KUKA KRL program: EPS_2_25862_MH07_A_20251016035156.src

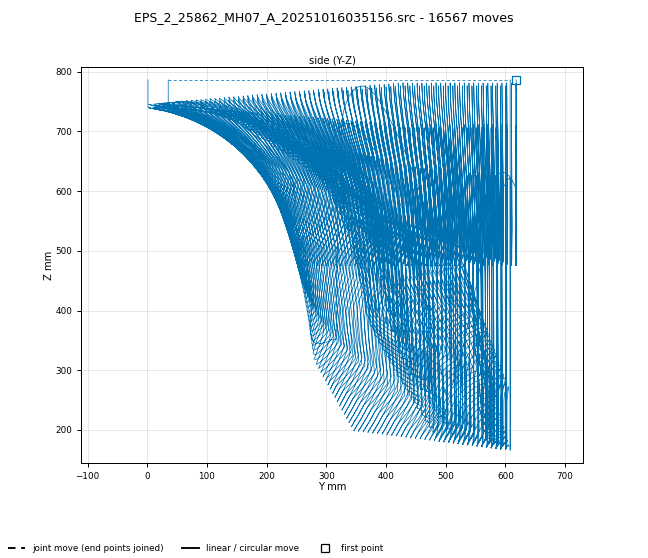
[picture p0: tool path of EPS_2_25862_MH07_A_20251016035156.src, 16567 of 16569 moves have a stored position in this frame; points joined in program order, loops and branches not executed]
&ACCESS RVP
&REL 4
&COMMENT QRS 19112012
&PARAM EDITMASK = *
DEF PART()
EXT BAS (BAS_COMMAND :IN,REAL :IN )
INT I
BAS (#INITMOV,0 )

;KUKA QRS Post kuka4.cps  Date:22-06-2017 !

File_ID=2887

QRS_PRE_INIT()

;Init var - Until changes are made in qrs_pre_init
Outlet_Square_prg=0
Inlet_1_Square_prg=0
Inlet_2_Square_prg=0
Inlet_3_Square_prg=0
Inlet_4_Square_prg=0
Inlet_5_Square_prg=0

Outlet_1={X 0.000, Y 425.000, Z 510.000, B 0.000, E1 0.000 }
Inlet_1={X 0.000, Y 529.170, Z 407.000, B 0.000, E1 90.000 }
Inlet_2={X 0.000, Y 425.000, Z 440.000, B 0.000, E1 163.000 }
Outlet_1_type=533
Inlet_1_type=299
Inlet_2_type=533
;QRS#1=Sidecore dimensions
;QRS#2=525-21" Concrete
;QRS#3=300-12" PVC SDR 35
;QRS#4=525-21" Concrete
;QRS#5=
;QRS#6=
;QRS#7=
;QRS#8=
;QRS#9=S306-32
;QRS#10=16M PSX
;QRS#11=S306-32
;QRS#12=
;QRS#13=
;QRS#14=
;QRS#15=
;QRS#16=1220x127x1143 3,75'
;QRS#17=EPS Height
;QRS#18=776,5
;QRS#19=*
;QRS#20= UPDATED VERSION 22-06-2017
;QRS#21=*
Outlet_Square=0250
Inlet_1_Square=0150
Inlet_2_Square=0250
Inlet_3_Square=0
Inlet_4_Square=0
Inlet_5_Square=0
Mill_Square=1
Outlet_Square_Prg=263
Inlet_1_Square_prg=206
Inlet_2_Square_prg=263

QRS_INIT()

$ADVANCE=5

; T1
PTP {E1 170.881,E2 170.881}
PTP {X 0,Y 617.976,A -85,B 0,C 180,E1 170.881,E2 170.881,E3 0,E4 0,E5 0,E6 0}
QRS_SPEED_INIT()
LIN {X 0,Y 617.976,Z 786.5,A -85,B 0,C 180,E1 170.881,E2 170.881,E3 0,E4 0,E5 0,E6 0} C_VEL
LIN {X 0,Y 617.976,Z 614.117,A -85,B 0,C 180,E1 170.881,E2 170.881} C_VEL
LIN {X 0,Y 617.976,Z 605.661,A -85,B 0,C 180,E1 170.881,E2 170.881} C_VEL
LIN {X 0,Y 617.953,Z 603.915,A -85,B 0,C 180,E1 171.157,E2 171.157} C_VEL
LIN {X 0,Y 617.982,Z 609.709,A -85,B 0,C 180,E1 172.119,E2 172.119} C_VEL
LIN {X 0,Y 617.938,Z 613.421,A -85,B 0,C 180,E1 172.818,E2 172.818} C_VEL
LIN {X 0,Y 617.912,Z 616.713,A -85,B 0,C 180,E1 173.515,E2 173.515} C_VEL
LIN {X 0,Y 617.958,Z 619.593,A -85,B 0,C 180,E1 174.213,E2 174.213} C_VEL
LIN {X 0,Y 617.989,Z 621.321,A -85,B 0,C 180,E1 174.678,E2 174.678} C_VEL
LIN {X 0,Y 617.915,Z 624.296,A -85,B 0,C 180,E1 175.605,E2 175.605} C_VEL
LIN {X 0,Y 617.888,Z 626.636,A -85,B 0,C 180,E1 176.531,E2 176.531} C_VEL
LIN {X 0,Y 617.975,Z 628.385,A -85,B 0,C 180,E1 177.457,E2 177.457} C_VEL
LIN {X 0,Y 617.924,Z 629.629,A -85,B 0,C 180,E1 178.382,E2 178.382} C_VEL
LIN {X 0,Y 617.892,Z 630.009,A -85,B 0,C 180,E1 178.844,E2 178.844} C_VEL
LIN {X 0,Y 617.918,Z 630.398,A -85,B 0,C 180,E1 179.769,E2 179.769} C_VEL
LIN {X 0,Y 617.987,Z 630.242,A -85,B 0,C 180,E1 180.693,E2 180.693} C_VEL
LIN {X 0,Y 617.941,Z 629.932,A -85,B 0,C 180,E1 181.156,E2 181.156} C_VEL
LIN {X 0,Y 617.883,Z 628.987,A -85,B 0,C 180,E1 182.08,E2 182.08} C_VEL
LIN {X 0,Y 617.888,Z 628.258,A -85,B 0,C 180,E1 182.543,E2 182.543} C_VEL
LIN {X 0,Y 617.984,Z 626.416,A -85,B 0,C 180,E1 183.468,E2 183.468} C_VEL
LIN {X 0,Y 617.908,Z 624.054,A -85,B 0,C 180,E1 184.395,E2 184.395} C_VEL
LIN {X 0,Y 617.895,Z 621.008,A -85,B 0,C 180,E1 185.323,E2 185.323} C_VEL
LIN {X 0,Y 617.935,Z 619.264,A -85,B 0,C 180,E1 185.787,E2 185.787} C_VEL
LIN {X 0,Y 617.983,Z 615.24,A -85,B 0,C 180,E1 186.716,E2 186.716} C_VEL
LIN {X 0,Y 617.925,Z 610.505,A -85,B 0,C 180,E1 187.649,E2 187.649} C_VEL
LIN {X 0,Y 617.962,Z 604.94,A -85,B 0,C 180,E1 188.595,E2 188.595} C_VEL
LIN {X 0,Y 618,Z 599.801,A -85,B 0,C 180,E1 189.355,E2 189.355} C_VEL
LIN {X 0,Y 617.956,Z 594.236,A -85,B 0,C 180,E1 190.089,E2 190.089} C_VEL
LIN {X 0,Y 617.957,Z 588.665,A -85,B 0,C 180,E1 190.75,E2 190.75} C_VEL
LIN {X 0,Y 617.996,Z 581.774,A -85,B 0,C 180,E1 191.486,E2 191.486} C_VEL
LIN {X 0,Y 617.98,Z 574.003,A -85,B 0,C 180,E1 192.224,E2 192.224} C_VEL
LIN {X 0,Y 617.981,Z 566.983,A -85,B 0,C 180,E1 192.815,E2 192.815} C_VEL
LIN {X 0,Y 618.01,Z 560.186,A -85,B 0,C 180,E1 193.334,E2 193.334} C_VEL
LIN {X 0,Y 618.026,Z 552.645,A -85,B 0,C 180,E1 193.853,E2 193.853} C_VEL
LIN {X 0,Y 618.025,Z 542.922,A -85,B 0,C 180,E1 194.449,E2 194.449} C_VEL
LIN {X 0,Y 617.99,Z 534.465,A -85,B 0,C 180,E1 194.898,E2 194.898} C_VEL
LIN {X 0,Y 618.023,Z 525.506,A -85,B 0,C 180,E1 195.313,E2 195.313} C_VEL
LIN {X 0,Y 618.026,Z 518.365,A -85,B 0,C 180,E1 195.605,E2 195.605} C_VEL
LIN {X 0,Y 617.977,Z 509.686,A -85,B 0,C 180,E1 195.915,E2 195.915} C_VEL
LIN {X 0,Y 617.998,Z 501.407,A -85,B 0,C 180,E1 196.165,E2 196.165} C_VEL
LIN {X 0,Y 618.025,Z 492.067,A -85,B 0,C 180,E1 196.398,E2 196.398} C_VEL
LIN {X 0,Y 617.952,Z 480.006,A -85,B 0,C 180,E1 196.626,E2 196.626} C_VEL
LIN {X 0,Y 617.88,Z 476.03,A -85,B 0,C 180,E1 196.691,E2 196.691} C_VEL
LIN {X 0,Y 618.007,Z 476.03,A -85,B 0,C 180,E1 196.801,E2 196.801} C_VEL
LIN {X 0,Y 617.96,Z 476.03,A -85,B 0,C 180,E1 200.048,E2 200.048} C_VEL
LIN {X 0,Y 617.455,Z 476.03,A -85,B 0,C 180,E1 202.548,E2 202.548} C_VEL
LIN {X 0,Y 617.918,Z 476.03,A -85,B 0,C 180,E1 205.056,E2 205.056} C_VEL
LIN {X 0,Y 617.406,Z 476.03,A -85,B 0,C 180,E1 207.66,E2 207.66} C_VEL
LIN {X 0,Y 617.848,Z 476.03,A -85,B 0,C 180,E1 210.28,E2 210.28} C_VEL
LIN {X 0,Y 617.31,Z 476.03,A -85,B 0,C 180,E1 213.027,E2 213.027} C_VEL
LIN {X 0,Y 617.797,Z 476.03,A -85,B 0,C 180,E1 215.799,E2 215.799} C_VEL
LIN {X 0,Y 617.573,Z 476.03,A -85,B 0,C 180,E1 218.099,E2 218.099} C_VEL
LIN {X 0,Y 617.553,Z 476.03,A -85,B 0,C 180,E1 218.722,E2 218.722} C_VEL
LIN {X 0,Y 617.792,Z 476.03,A -85,B 0,C 180,E1 221.731,E2 221.731} C_VEL
LIN {X 0,Y 617.879,Z 476.03,A -85,B 0,C 180,E1 225.099,E2 225.099} C_VEL
LIN {X 0,Y 617.456,Z 476.03,A -85,B 0,C 180,E1 228.308,E2 228.308} C_VEL
LIN {X 0,Y 617.797,Z 476.03,A -85,B 0,C 180,E1 231.296,E2 231.296} C_VEL
LIN {X 0,Y 617.723,Z 476.03,A -85,B 0,C 180,E1 235.802,E2 235.802} C_VEL
LIN {X 0,Y 617.906,Z 476.03,A -85,B 0,C 180,E1 237.009,E2 237.009} C_VEL
LIN {X 0,Y 617.905,Z 476.03,A -85,B 0,C 180,E1 240.133,E2 240.133} C_VEL
LIN {X 0,Y 617.607,Z 476.03,A -85,B 0,C 180,E1 240.837,E2 240.837} C_VEL
LIN {X 0,Y 617.093,Z 483.978,A -85,B 0,C 180,E1 241.034,E2 241.034} C_VEL
LIN {X 0,Y 617.595,Z 516.166,A -85,B 0,C 180,E1 241.478,E2 241.478} C_VEL
LIN {X 0,Y 617.687,Z 536.067,A -85,B 0,C 180,E1 241.783,E2 241.783} C_VEL
LIN {X 0,Y 617.745,Z 546.864,A -85,B 0,C 180,E1 242.005,E2 242.005} C_VEL
LIN {X 0,Y 617.719,Z 563.319,A -85,B 0,C 180,E1 242.427,E2 242.427} C_VEL
LIN {X 0,Y 617.856,Z 576.645,A -85,B 0,C 180,E1 242.85,E2 242.85} C_VEL
LIN {X 0,Y 617.886,Z 587.938,A -85,B 0,C 180,E1 243.257,E2 243.257} C_VEL
LIN {X 0,Y 617.754,Z 601.563,A -85,B 0,C 180,E1 243.815,E2 243.815} C_VEL
LIN {X 0,Y 617.879,Z 613.583,A -85,B 0,C 180,E1 244.383,E2 244.383} C_VEL
LIN {X 0,Y 617.884,Z 625.767,A -85,B 0,C 180,E1 245.021,E2 245.021} C_VEL
LIN {X 0,Y 617.847,Z 637.421,A -85,B 0,C 180,E1 245.696,E2 245.696} C_VEL
LIN {X 0,Y 617.908,Z 648.138,A -85,B 0,C 180,E1 246.38,E2 246.38} C_VEL
LIN {X 0,Y 617.924,Z 659.39,A -85,B 0,C 180,E1 247.168,E2 247.168} C_VEL
LIN {X 0,Y 617.915,Z 669.503,A -85,B 0,C 180,E1 247.938,E2 247.938} C_VEL
LIN {X 0,Y 617.885,Z 680.645,A -85,B 0,C 180,E1 248.869,E2 248.869} C_VEL
LIN {X 0,Y 617.922,Z 690.764,A -85,B 0,C 180,E1 249.797,E2 249.797} C_VEL
LIN {X 0,Y 617.932,Z 699.516,A -85,B 0,C 180,E1 250.667,E2 250.667} C_VEL
LIN {X 0,Y 617.881,Z 706.64,A -85,B 0,C 180,E1 251.422,E2 251.422} C_VEL
LIN {X 0,Y 617.901,Z 715.015,A -85,B 0,C 180,E1 252.391,E2 252.391} C_VEL
LIN {X 0,Y 617.982,Z 723.19,A -85,B 0,C 180,E1 253.428,E2 253.428} C_VEL
LIN {X 0,Y 617.837,Z 731.707,A -85,B 0,C 180,E1 254.61,E2 254.61} C_VEL
LIN {X 0,Y 617.891,Z 738.767,A -85,B 0,C 180,E1 255.697,E2 255.697} C_VEL
LIN {X 0,Y 617.963,Z 744.12,A -85,B 0,C 180,E1 256.591,E2 256.591} C_VEL
LIN {X 0,Y 617.785,Z 750.562,A -85,B 0,C 180,E1 257.772,E2 257.772} C_VEL
LIN {X 0,Y 617.806,Z 756.245,A -85,B 0,C 180,E1 258.953,E2 258.953} C_VEL
LIN {X 0,Y 617.974,Z 760.457,A -85,B 0,C 180,E1 259.949,E2 259.949} C_VEL
LIN {X 0,Y 617.8,Z 765.453,A -85,B 0,C 180,E1 261.249,E2 261.249} C_VEL
LIN {X 0,Y 617.8,Z 769.018,A -85,B 0,C 180,E1 262.35,E2 262.35} C_VEL
LIN {X 0,Y 617.952,Z 772.841,A -85,B 0,C 180,E1 263.748,E2 263.748} C_VEL
LIN {X 0,Y 617.735,Z 775.904,A -85,B 0,C 180,E1 265.14,E2 265.14} C_VEL
LIN {X 0,Y 617.832,Z 778.096,A -85,B 0,C 180,E1 266.531,E2 266.531} C_VEL
LIN {X 0,Y 617.874,Z 779.552,A -85,B 0,C 180,E1 267.919,E2 267.919} C_VEL
LIN {X 0,Y 617.748,Z 780.216,A -85,B 0,C 180,E1 268.844,E2 268.844} C_VEL
LIN {X 0,Y 617.993,Z 780.149,A -85,B 0,C 180,E1 271.155,E2 271.155} C_VEL
LIN {X 0,Y 617.921,Z 779.182,A -85,B 0,C 180,E1 272.543,E2 272.543} C_VEL
LIN {X 0,Y 617.992,Z 778.053,A -85,B 0,C 180,E1 273.468,E2 273.468} C_VEL
LIN {X 0,Y 617.764,Z 775.897,A -85,B 0,C 180,E1 274.86,E2 274.86} C_VEL
LIN {X 0,Y 617.792,Z 772.883,A -85,B 0,C 180,E1 276.253,E2 276.253} C_VEL
LIN {X 0,Y 617.96,Z 770.333,A -85,B 0,C 180,E1 277.182,E2 277.182} C_VEL
LIN {X 0,Y 617.863,Z 767.502,A -85,B 0,C 180,E1 278.116,E2 278.116} C_VEL
LIN {X 0,Y 617.789,Z 765.164,A -85,B 0,C 180,E1 278.829,E2 278.829} C_VEL
LIN {X 0,Y 617.862,Z 760.497,A -85,B 0,C 180,E1 280.05,E2 280.05} C_VEL
LIN {X 0,Y 617.967,Z 756.211,A -85,B 0,C 180,E1 281.044,E2 281.044} C_VEL
LIN {X 0,Y 617.792,Z 750.562,A -85,B 0,C 180,E1 282.227,E2 282.227} C_VEL
LIN {X 0,Y 617.814,Z 744.15,A -85,B 0,C 180,E1 283.412,E2 283.412} C_VEL
LIN {X 0,Y 617.958,Z 736.918,A -85,B 0,C 180,E1 284.6,E2 284.6} C_VEL
LIN {X 0,Y 617.812,Z 729.351,A -85,B 0,C 180,E1 285.734,E2 285.734} C_VEL
LIN {X 0,Y 617.84,Z 722.479,A -85,B 0,C 180,E1 286.674,E2 286.674} C_VEL
LIN {X 0,Y 617.977,Z 713.931,A -85,B 0,C 180,E1 287.734,E2 287.734} C_VEL
LIN {X 0,Y 617.889,Z 704.471,A -85,B 0,C 180,E1 288.81,E2 288.81} C_VEL
LIN {X 0,Y 617.892,Z 695.989,A -85,B 0,C 180,E1 289.695,E2 289.695} C_VEL
LIN {X 0,Y 617.937,Z 687.527,A -85,B 0,C 180,E1 290.511,E2 290.511} C_VEL
LIN {X 0,Y 617.894,Z 677.03,A -85,B 0,C 180,E1 291.44,E2 291.44} C_VEL
LIN {X 0,Y 617.882,Z 667.492,A -85,B 0,C 180,E1 292.219,E2 292.219} C_VEL
LIN {X 0,Y 617.9,Z 657.417,A -85,B 0,C 180,E1 292.976,E2 292.976} C_VEL
LIN {X 0,Y 617.911,Z 645.135,A -85,B 0,C 180,E1 293.813,E2 293.813} C_VEL
LIN {X 0,Y 617.904,Z 633.893,A -85,B 0,C 180,E1 294.512,E2 294.512} C_VEL
LIN {X 0,Y 617.836,Z 622.881,A -85,B 0,C 180,E1 295.139,E2 295.139} C_VEL
LIN {X 0,Y 617.892,Z 610.287,A -85,B 0,C 180,E1 295.776,E2 295.776} C_VEL
LIN {X 0,Y 617.876,Z 597.865,A -85,B 0,C 180,E1 296.34,E2 296.34} C_VEL
LIN {X 0,Y 617.703,Z 584.662,A -85,B 0,C 180,E1 296.873,E2 296.873} C_VEL
LIN {X 0,Y 617.832,Z 571.391,A -85,B 0,C 180,E1 297.323,E2 297.323} C_VEL
LIN {X 0,Y 617.741,Z 558.539,A -85,B 0,C 180,E1 297.705,E2 297.705} C_VEL
LIN {X 0,Y 617.713,Z 550.591,A -85,B 0,C 180,E1 297.907,E2 297.907} C_VEL
LIN {X 0,Y 617.901,Z 535.737,A -85,B 0,C 180,E1 298.213,E2 298.213} C_VEL
LIN {X 0,Y 617.756,Z 515.651,A -85,B 0,C 180,E1 298.521,E2 298.521} C_VEL
LIN {X 0,Y 617.026,Z 476.03,A -85,B 0,C 180,E1 299.084,E2 299.084} C_VEL
LIN {X 0,Y 618.06,Z 476.03,A -85,B 0,C 180,E1 299.464,E2 299.464} C_VEL
LIN {X 0,Y 618.044,Z 476.03,A -85,B 0,C 180,E1 300.269,E2 300.269} C_VEL
LIN {X 0,Y 617.372,Z 476.03,A -85,B 0,C 180,E1 304.15,E2 304.15} C_VEL
LIN {X 0,Y 617.829,Z 476.03,A -85,B 0,C 180,E1 305.797,E2 305.797} C_VEL
LIN {X 0,Y 617.555,Z 476.03,A -85,B 0,C 180,E1 308.721,E2 308.721} C_VEL
LIN {X 0,Y 617.763,Z 476.03,A -85,B 0,C 180,E1 311.733,E2 311.733} C_VEL
LIN {X 0,Y 617.85,Z 476.03,A -85,B 0,C 180,E1 315.097,E2 315.097} C_VEL
LIN {X 0,Y 617.449,Z 476.03,A -85,B 0,C 180,E1 318.308,E2 318.308} C_VEL
LIN {X 0,Y 617.792,Z 476.03,A -85,B 0,C 180,E1 321.296,E2 321.296} C_VEL
LIN {X 0,Y 617.737,Z 476.03,A -85,B 0,C 180,E1 325.799,E2 325.799} C_VEL
LIN {X 0,Y 617.89,Z 476.03,A -85,B 0,C 180,E1 327.008,E2 327.008} C_VEL
LIN {X 0,Y 617.613,Z 476.03,A -85,B 0,C 180,E1 330.18,E2 330.18} C_VEL
LIN {X 0,Y 617.623,Z 476.03,A -85,B 0,C 180,E1 332.351,E2 332.351} C_VEL
LIN {X 0,Y 617.512,Z 476.03,A -85,B 0,C 180,E1 335.243,E2 335.243} C_VEL
LIN {X 0,Y 617.738,Z 476.03,A -85,B 0,C 180,E1 337.463,E2 337.463} C_VEL
LIN {X 0,Y 617.768,Z 476.03,A -85,B 0,C 180,E1 341.452,E2 341.452} C_VEL
LIN {X 0,Y 617.981,Z 476.03,A -85,B 0,C 180,E1 342.394,E2 342.394} C_VEL
LIN {X 0,Y 618.01,Z 476.03,A -85,B 0,C 180,E1 347.185,E2 347.185} C_VEL
LIN {X 0,Y 617.973,Z 476.03,A -85,B 0,C 180,E1 351.885,E2 351.885} C_VEL
LIN {X 0,Y 618.058,Z 476.03,A -85,B 0,C 180,E1 356.532,E2 356.532} C_VEL
LIN {X 0,Y 618.062,Z 476.03,A -85,B 0,C 180,E1 361.155,E2 361.155} C_VEL
LIN {X 0,Y 618.025,Z 476.03,A -85,B 0,C 180,E1 365.786,E2 365.786} C_VEL
LIN {X 0,Y 618.005,Z 476.03,A -85,B 0,C 180,E1 370.456,E2 370.456} C_VEL
LIN {X 0,Y 617.94,Z 476.03,A -85,B 0,C 180,E1 375.198,E2 375.198} C_VEL
LIN {X 0,Y 617.959,Z 476.03,A -85,B 0,C 180,E1 380.048,E2 380.048} C_VEL
LIN {X 0,Y 617.477,Z 476.03,A -85,B 0,C 180,E1 382.547,E2 382.547} C_VEL
LIN {X 0,Y 617.928,Z 476.03,A -85,B 0,C 180,E1 385.055,E2 385.055} C_VEL
LIN {X 0,Y 617.434,Z 476.03,A -85,B 0,C 180,E1 387.658,E2 387.658} C_VEL
LIN {X 0,Y 617.899,Z 476.03,A -85,B 0,C 180,E1 390.277,E2 390.277} C_VEL
LIN {X 0,Y 617.363,Z 476.03,A -85,B 0,C 180,E1 393.024,E2 393.024} C_VEL
LIN {X 0,Y 617.83,Z 476.03,A -85,B 0,C 180,E1 395.797,E2 395.797} C_VEL
LIN {X 0,Y 617.922,Z 476.03,A -85,B 0,C 180,E1 398.694,E2 398.694} C_VEL
LIN {X 0,Y 617.441,Z 476.03,A -85,B 0,C 180,E1 401.76,E2 401.76} C_VEL
LIN {X 0,Y 617.884,Z 476.03,A -85,B 0,C 180,E1 404.9,E2 404.9} C_VEL
LIN {X 0,Y 617.788,Z 476.03,A -85,B 0,C 180,E1 408.273,E2 408.273} C_VEL
LIN {X 0,Y 617.543,Z 476.03,A -85,B 0,C 180,E1 411.278,E2 411.278} C_VEL
LIN {X 0,Y 617.56,Z 476.03,A -85,B 0,C 180,E1 411.902,E2 411.902} C_VEL
LIN {X 0,Y 617.774,Z 476.03,A -85,B 0,C 180,E1 414.199,E2 414.199} C_VEL
LIN {X 0,Y 617.311,Z 476.03,A -85,B 0,C 180,E1 416.973,E2 416.973} C_VEL
LIN {X 0,Y 617.85,Z 476.03,A -85,B 0,C 180,E1 419.72,E2 419.72} C_VEL
LIN {X 0,Y 617.406,Z 476.03,A -85,B 0,C 180,E1 422.341,E2 422.341} C_VEL
LIN {X 0,Y 617.916,Z 476.03,A -85,B 0,C 180,E1 424.944,E2 424.944} C_VEL
LIN {X 0,Y 617.454,Z 476.03,A -85,B 0,C 180,E1 427.452,E2 427.452} C_VEL
LIN {X 0,Y 617.947,Z 476.03,A -85,B 0,C 180,E1 429.952,E2 429.952} C_VEL
LIN {X 0,Y 617.716,Z 476.03,A -85,B 0,C 180,E1 432.386,E2 432.386} C_VEL
LIN {X 0,Y 617.639,Z 476.03,A -85,B 0,C 180,E1 434.795,E2 434.795} C_VEL
LIN {X 0,Y 617.816,Z 476.03,A -85,B 0,C 180,E1 437.834,E2 437.834} C_VEL
LIN {X 0,Y 617.958,Z 476.03,A -85,B 0,C 180,E1 438.667,E2 438.667} C_VEL
LIN {X 0,Y 617.118,Z 476.03,A -85,B 0,C 180,E1 438.912,E2 438.912} C_VEL
LIN {X 0,Y 617.601,Z 477.618,A -85,B 0,C 180,E1 438.969,E2 438.969} C_VEL
LIN {X 0,Y 617.721,Z 492.547,A -85,B 0,C 180,E1 439.358,E2 439.358} C_VEL
LIN {X 0,Y 617.858,Z 505.819,A -85,B 0,C 180,E1 439.776,E2 439.776} C_VEL
LIN {X 0,Y 617.814,Z 518.782,A -85,B 0,C 180,E1 440.243,E2 440.243} C_VEL
LIN {X 0,Y 617.844,Z 529.089,A -85,B 0,C 180,E1 440.664,E2 440.664} C_VEL
LIN {X 0,Y 617.915,Z 543.28,A -85,B 0,C 180,E1 441.324,E2 441.324} C_VEL
LIN {X 0,Y 617.87,Z 556.214,A -85,B 0,C 180,E1 442.001,E2 442.001} C_VEL
LIN {X 0,Y 617.891,Z 568.182,A -85,B 0,C 180,E1 442.701,E2 442.701} C_VEL
LIN {X 0,Y 617.899,Z 579.063,A -85,B 0,C 180,E1 443.399,E2 443.399} C_VEL
LIN {X 0,Y 617.912,Z 590.579,A -85,B 0,C 180,E1 444.213,E2 444.213} C_VEL
LIN {X 0,Y 617.9,Z 601.106,A -85,B 0,C 180,E1 445.025,E2 445.025} C_VEL
LIN {X 0,Y 617.886,Z 610.785,A -85,B 0,C 180,E1 445.837,E2 445.837} C_VEL
LIN {X 0,Y 617.945,Z 619.692,A -85,B 0,C 180,E1 446.648,E2 446.648} C_VEL
LIN {X 0,Y 617.931,Z 629.056,A -85,B 0,C 180,E1 447.573,E2 447.573} C_VEL
LIN {X 0,Y 617.868,Z 637.688,A -85,B 0,C 180,E1 448.498,E2 448.498} C_VEL
LIN {X 0,Y 617.917,Z 644.688,A -85,B 0,C 180,E1 449.307,E2 449.307} C_VEL
LIN {X 0,Y 617.934,Z 653.784,A -85,B 0,C 180,E1 450.462,E2 450.462} C_VEL
LIN {X 0,Y 617.824,Z 660.536,A -85,B 0,C 180,E1 451.387,E2 451.387} C_VEL
LIN {X 0,Y 617.897,Z 668.115,A -85,B 0,C 180,E1 452.543,E2 452.543} C_VEL
LIN {X 0,Y 617.949,Z 673.665,A -85,B 0,C 180,E1 453.469,E2 453.469} C_VEL
LIN {X 0,Y 617.77,Z 681.208,A -85,B 0,C 180,E1 454.86,E2 454.86} C_VEL
LIN {X 0,Y 617.862,Z 686.708,A -85,B 0,C 180,E1 456.02,E2 456.02} C_VEL
LIN {X 0,Y 617.963,Z 689.656,A -85,B 0,C 180,E1 456.717,E2 456.717} C_VEL
LIN {X 0,Y 617.838,Z 693.365,A -85,B 0,C 180,E1 457.65,E2 457.65} C_VEL
LIN {X 0,Y 617.773,Z 696.469,A -85,B 0,C 180,E1 458.508,E2 458.508} C_VEL
LIN {X 0,Y 617.884,Z 700.002,A -85,B 0,C 180,E1 459.641,E2 459.641} C_VEL
LIN {X 0,Y 617.973,Z 702.167,A -85,B 0,C 180,E1 460.456,E2 460.456} C_VEL
LIN {X 0,Y 617.795,Z 704.937,A -85,B 0,C 180,E1 461.637,E2 461.637} C_VEL
LIN {X 0,Y 617.827,Z 707.092,A -85,B 0,C 180,E1 462.819,E2 462.819} C_VEL
LIN {X 0,Y 617.971,Z 708.672,A -85,B 0,C 180,E1 464.004,E2 464.004} C_VEL
LIN {X 0,Y 617.751,Z 709.818,A -85,B 0,C 180,E1 465.203,E2 465.203} C_VEL
LIN {X 0,Y 617.724,Z 710.336,A -85,B 0,C 180,E1 466.313,E2 466.313} C_VEL
LIN {X 0,Y 617.943,Z 710.275,A -85,B 0,C 180,E1 467.607,E2 467.607} C_VEL
LIN {X 0,Y 617.891,Z 709.834,A -85,B 0,C 180,E1 468.632,E2 468.632} C_VEL
LIN {X 0,Y 617.915,Z 708.516,A -85,B 0,C 180,E1 470.05,E2 470.05} C_VEL
LIN {X 0,Y 617.852,Z 706.755,A -85,B 0,C 180,E1 471.287,E2 471.287} C_VEL
LIN {X 0,Y 617.777,Z 705.727,A -85,B 0,C 180,E1 471.911,E2 471.911} C_VEL
LIN {X 0,Y 617.771,Z 703.259,A -85,B 0,C 180,E1 473.047,E2 473.047} C_VEL
LIN {X 0,Y 617.987,Z 699.619,A -85,B 0,C 180,E1 474.399,E2 474.399} C_VEL
LIN {X 0,Y 617.775,Z 695.478,A -85,B 0,C 180,E1 475.702,E2 475.702} C_VEL
LIN {X 0,Y 617.81,Z 690.576,A -85,B 0,C 180,E1 476.99,E2 476.99} C_VEL
LIN {X 0,Y 617.965,Z 685.729,A -85,B 0,C 180,E1 478.104,E2 478.104} C_VEL
LIN {X 0,Y 617.824,Z 680.253,A -85,B 0,C 180,E1 479.241,E2 479.241} C_VEL
LIN {X 0,Y 617.876,Z 673.662,A -85,B 0,C 180,E1 480.446,E2 480.446} C_VEL
LIN {X 0,Y 617.958,Z 666.474,A -85,B 0,C 180,E1 481.621,E2 481.621} C_VEL
LIN {X 0,Y 617.833,Z 658.598,A -85,B 0,C 180,E1 482.791,E2 482.791} C_VEL
LIN {X 0,Y 617.908,Z 651.168,A -85,B 0,C 180,E1 483.79,E2 483.79} C_VEL
LIN {X 0,Y 617.983,Z 644.312,A -85,B 0,C 180,E1 484.645,E2 484.645} C_VEL
LIN {X 0,Y 617.871,Z 634.198,A -85,B 0,C 180,E1 485.795,E2 485.795} C_VEL
LIN {X 0,Y 617.907,Z 625.412,A -85,B 0,C 180,E1 486.706,E2 486.706} C_VEL
LIN {X 0,Y 617.936,Z 616.132,A -85,B 0,C 180,E1 487.591,E2 487.591} C_VEL
LIN {X 0,Y 617.914,Z 608.131,A -85,B 0,C 180,E1 488.304,E2 488.304} C_VEL
LIN {X 0,Y 617.888,Z 597.463,A -85,B 0,C 180,E1 489.176,E2 489.176} C_VEL
LIN {X 0,Y 617.868,Z 587.152,A -85,B 0,C 180,E1 489.95,E2 489.95} C_VEL
LIN {X 0,Y 617.904,Z 576.246,A -85,B 0,C 180,E1 490.699,E2 490.699} C_VEL
LIN {X 0,Y 617.902,Z 564.345,A -85,B 0,C 180,E1 491.441,E2 491.441} C_VEL
LIN {X 0,Y 617.813,Z 551.969,A -85,B 0,C 180,E1 492.142,E2 492.142} C_VEL
LIN {X 0,Y 617.871,Z 540.321,A -85,B 0,C 180,E1 492.731,E2 492.731} C_VEL
LIN {X 0,Y 617.851,Z 528.459,A -85,B 0,C 180,E1 493.271,E2 493.271} C_VEL
LIN {X 0,Y 617.723,Z 515.883,A -85,B 0,C 180,E1 493.784,E2 493.784} C_VEL
LIN {X 0,Y 617.856,Z 501.446,A -85,B 0,C 180,E1 494.275,E2 494.275} C_VEL
LIN {X 0,Y 617.787,Z 488.688,A -85,B 0,C 180,E1 494.654,E2 494.654} C_VEL
LIN {X 0,Y 617.518,Z 476.03,A -85,B 0,C 180,E1 494.988,E2 494.988} C_VEL
LIN {X 0,Y 618.002,Z 476.03,A -85,B 0,C 180,E1 495.111,E2 495.111} C_VEL
LIN {X 0,Y 617.354,Z 476.03,A -85,B 0,C 180,E1 498.318,E2 498.318} C_VEL
LIN {X 0,Y 617.788,Z 476.03,A -85,B 0,C 180,E1 501.296,E2 501.296} C_VEL
LIN {X 0,Y 617.711,Z 476.03,A -85,B 0,C 180,E1 505.803,E2 505.803} C_VEL
LIN {X 0,Y 617.878,Z 476.03,A -85,B 0,C 180,E1 507.007,E2 507.007} C_VEL
LIN {X 0,Y 618.031,Z 476.03,A -85,B 0,C 180,E1 511.492,E2 511.492} C_VEL
LIN {X 0,Y 617.378,Z 476.03,A -85,B 0,C 180,E1 515.271,E2 515.271} C_VEL
LIN {X 0,Y 617.928,Z 476.03,A -85,B 0,C 180,E1 517.47,E2 517.47} C_VEL
LIN {X 0,Y 618.059,Z 476.03,A -85,B 0,C 180,E1 522.8,E2 522.8} C_VEL
LIN {X 0,Y 616.384,Z 476.03,A -85,B 0,C 180,E1 523.155,E2 523.155} C_VEL
LIN {X 0,Y 616.161,Z 476.1,A -85,B 0,C 180,E1 523.179,E2 523.179} C_VEL
LIN {X 0,Y 617.345,Z 479.078,A -85,B 0,C 180,E1 523.254,E2 523.254} C_VEL
LIN {X 0,Y 617.909,Z 482.221,A -85,B 0,C 180,E1 523.316,E2 523.316} C_VEL
LIN {X 0,Y 617.987,Z 492.727,A -85,B 0,C 180,E1 523.526,E2 523.526} C_VEL
LIN {X 0,Y 617.947,Z 501.655,A -85,B 0,C 180,E1 523.751,E2 523.751} C_VEL
LIN {X 0,Y 617.991,Z 509.87,A -85,B 0,C 180,E1 524.001,E2 524.001} C_VEL
LIN {X 0,Y 617.968,Z 518.24,A -85,B 0,C 180,E1 524.299,E2 524.299} C_VEL
LIN {X 0,Y 617.97,Z 524.958,A -85,B 0,C 180,E1 524.572,E2 524.572} C_VEL
LIN {X 0,Y 618.003,Z 533.233,A -85,B 0,C 180,E1 524.953,E2 524.953} C_VEL
LIN {X 0,Y 618.025,Z 541.829,A -85,B 0,C 180,E1 525.402,E2 525.402} C_VEL
LIN {X 0,Y 617.985,Z 551.76,A -85,B 0,C 180,E1 525.997,E2 525.997} C_VEL
LIN {X 0,Y 618,Z 559.381,A -85,B 0,C 180,E1 526.518,E2 526.518} C_VEL
LIN {X 0,Y 618.006,Z 566.245,A -85,B 0,C 180,E1 527.037,E2 527.037} C_VEL
LIN {X 0,Y 618.001,Z 573.331,A -85,B 0,C 180,E1 527.629,E2 527.629} C_VEL
LIN {X 0,Y 617.98,Z 581.22,A -85,B 0,C 180,E1 528.367,E2 528.367} C_VEL
LIN {X 0,Y 617.981,Z 586.842,A -85,B 0,C 180,E1 528.956,E2 528.956} C_VEL
LIN {X 0,Y 618.011,Z 591.964,A -85,B 0,C 180,E1 529.544,E2 529.544} C_VEL
LIN {X 0,Y 617.972,Z 597.992,A -85,B 0,C 180,E1 530.31,E2 530.31} C_VEL
LIN {X 0,Y 617.938,Z 603.365,A -85,B 0,C 180,E1 531.075,E2 531.075} C_VEL
LIN {X 0,Y 617.953,Z 603.915,A -85,B 0,C 180,E1 531.157,E2 531.157} C_VEL
LIN {X 0,Y 614.025,Z 612.896,A -85,B 0,C 180,E1 532.531,E2 532.531} C_VEL
LIN {X 0,Y 610.136,Z 619.876,A -85,B 0,C 180,E1 533.98,E2 533.98} C_VEL
LIN {X 0,Y 610.076,Z 627.528,A -85,B 0,C 180,E1 536.441,E2 536.441} C_VEL
LIN {X 0,Y 610.102,Z 630.881,A -85,B 0,C 180,E1 538.576,E2 538.576} C_VEL
LIN {X 0,Y 610.104,Z 630.818,A -85,B 0,C 180,E1 541.42,E2 541.42} C_VEL
LIN {X 0,Y 610.115,Z 625.509,A -85,B 0,C 180,E1 544.267,E2 544.267} C_VEL
LIN {X 0,Y 610.138,Z 614.506,A -85,B 0,C 180,E1 547.125,E2 547.125} C_VEL
LIN {X 0,Y 610.2,Z 597.879,A -85,B 0,C 180,E1 549.819,E2 549.819} C_VEL
LIN {X 0,Y 610.219,Z 576.647,A -85,B 0,C 180,E1 552.172,E2 552.172} C_VEL
LIN {X 0,Y 610.331,Z 550.663,A -85,B 0,C 180,E1 554.177,E2 554.177} C_VEL
LIN {X 0,Y 610.405,Z 521.112,A -85,B 0,C 180,E1 555.702,E2 555.702} C_VEL
LIN {X 0,Y 610.453,Z 489.709,A -85,B 0,C 180,E1 556.662,E2 556.662} C_VEL
LIN {X 0,Y 610.085,Z 476.03,A -85,B 0,C 180,E1 556.951,E2 556.951} C_VEL
LIN {X 0,Y 609.583,Z 476.03,A -85,B 0,C 180,E1 561.871,E2 561.871} C_VEL
LIN {X 0,Y 610.001,Z 476.03,A -85,B 0,C 180,E1 564.954,E2 564.954} C_VEL
LIN {X 0,Y 609.766,Z 476.03,A -85,B 0,C 180,E1 569.772,E2 569.772} C_VEL
LIN {X 0,Y 609.713,Z 476.03,A -85,B 0,C 180,E1 576.578,E2 576.578} C_VEL
LIN {X 0,Y 609.798,Z 476.03,A -85,B 0,C 180,E1 582.091,E2 582.091} C_VEL
LIN {X 0,Y 609.521,Z 476.03,A -85,B 0,C 180,E1 587.878,E2 587.878} C_VEL
LIN {X 0,Y 609.49,Z 476.03,A -85,B 0,C 180,E1 592.642,E2 592.642} C_VEL
LIN {X 0,Y 609.897,Z 476.03,A -85,B 0,C 180,E1 597.562,E2 597.562} C_VEL
LIN {X 0,Y 609.828,Z 476.03,A -85,B 0,C 180,E1 600.533,E2 600.533} C_VEL
LIN {X 0,Y 610.755,Z 548.666,A -85,B 0,C 180,E1 601.697,E2 601.697} C_VEL
LIN {X 0,Y 610.747,Z 588.608,A -85,B 0,C 180,E1 602.946,E2 602.946} C_VEL
LIN {X 0,Y 610.579,Z 625.307,A -85,B 0,C 180,E1 604.674,E2 604.674} C_VEL
LIN {X 0,Y 610.427,Z 661.111,A -85,B 0,C 180,E1 607.004,E2 607.004} C_VEL
LIN {X 0,Y 610.29,Z 692.229,A -85,B 0,C 180,E1 609.675,E2 609.675} C_VEL
LIN {X 0,Y 610.174,Z 719.223,A -85,B 0,C 180,E1 612.676,E2 612.676} C_VEL
LIN {X 0,Y 610.128,Z 742.058,A -85,B 0,C 180,E1 615.997,E2 615.997} C_VEL
LIN {X 0,Y 610.103,Z 760.364,A -85,B 0,C 180,E1 619.634,E2 619.634} C_VEL
LIN {X 0,Y 610.018,Z 772.184,A -85,B 0,C 180,E1 623.084,E2 623.084} C_VEL
LIN {X 0,Y 609.94,Z 777.931,A -85,B 0,C 180,E1 625.729,E2 625.729} C_VEL
LIN {X 0,Y 609.966,Z 781.082,A -85,B 0,C 180,E1 628.577,E2 628.577} C_VEL
LIN {X 0,Y 610.143,Z 781.082,A -85,B 0,C 180,E1 631.422,E2 631.422} C_VEL
LIN {X 0,Y 609.934,Z 776.726,A -85,B 0,C 180,E1 634.984,E2 634.984} C_VEL
LIN {X 0,Y 609.991,Z 767.209,A -85,B 0,C 180,E1 638.565,E2 638.565} C_VEL
LIN {X 0,Y 609.997,Z 752.077,A -85,B 0,C 180,E1 642.18,E2 642.18} C_VEL
LIN {X 0,Y 610.074,Z 731.595,A -85,B 0,C 180,E1 645.652,E2 645.652} C_VEL
LIN {X 0,Y 610.218,Z 705.456,A -85,B 0,C 180,E1 648.957,E2 648.957} C_VEL
LIN {X 0,Y 610.316,Z 675.52,A -85,B 0,C 180,E1 651.847,E2 651.847} C_VEL
LIN {X 0,Y 610.516,Z 643.09,A -85,B 0,C 180,E1 654.252,E2 654.252} C_VEL
LIN {X 0,Y 610.675,Z 608.046,A -85,B 0,C 180,E1 656.209,E2 656.209} C_VEL
LIN {X 0,Y 610.755,Z 571.097,A -85,B 0,C 180,E1 657.676,E2 657.676} C_VEL
LIN {X 0,Y 610.949,Z 534.061,A -85,B 0,C 180,E1 658.595,E2 658.595} C_VEL
LIN {X 0,Y 609.927,Z 476.03,A -85,B 0,C 180,E1 659.461,E2 659.461} C_VEL
LIN {X 0,Y 609.726,Z 476.03,A -85,B 0,C 180,E1 666.583,E2 666.583} C_VEL
LIN {X 0,Y 609.769,Z 476.03,A -85,B 0,C 180,E1 672.1,E2 672.1} C_VEL
LIN {X 0,Y 609.507,Z 476.03,A -85,B 0,C 180,E1 677.884,E2 677.884} C_VEL
LIN {X 0,Y 609.49,Z 476.03,A -85,B 0,C 180,E1 682.651,E2 682.651} C_VEL
LIN {X 0,Y 609.827,Z 476.03,A -85,B 0,C 180,E1 687.583,E2 687.583} C_VEL
LIN {X 0,Y 609.66,Z 476.03,A -85,B 0,C 180,E1 691.849,E2 691.849} C_VEL
LIN {X 0,Y 609.667,Z 476.03,A -85,B 0,C 180,E1 696.765,E2 696.765} C_VEL
LIN {X 0,Y 609.978,Z 476.03,A -85,B 0,C 180,E1 702.674,E2 702.674} C_VEL
LIN {X 0,Y 610.065,Z 476.03,A -85,B 0,C 180,E1 707.096,E2 707.096} C_VEL
LIN {X 0,Y 609.778,Z 476.03,A -85,B 0,C 180,E1 712.871,E2 712.871} C_VEL
LIN {X 0,Y 609.933,Z 476.03,A -85,B 0,C 180,E1 717.157,E2 717.157} C_VEL
LIN {X 0,Y 610.048,Z 476.03,A -85,B 0,C 180,E1 721.424,E2 721.424} C_VEL
LIN {X 0,Y 609.799,Z 476.03,A -85,B 0,C 180,E1 726.692,E2 726.692} C_VEL
LIN {X 0,Y 609.752,Z 476.03,A -85,B 0,C 180,E1 731.46,E2 731.46} C_VEL
LIN {X 0,Y 609.797,Z 476.03,A -85,B 0,C 180,E1 735.852,E2 735.852} C_VEL
LIN {X 0,Y 609.94,Z 476.03,A -85,B 0,C 180,E1 740.337,E2 740.337} C_VEL
LIN {X 0,Y 610.003,Z 476.03,A -85,B 0,C 180,E1 744.959,E2 744.959} C_VEL
LIN {X 0,Y 609.821,Z 476.03,A -85,B 0,C 180,E1 749.774,E2 749.774} C_VEL
LIN {X 0,Y 609.803,Z 476.03,A -85,B 0,C 180,E1 756.577,E2 756.577} C_VEL
LIN {X 0,Y 609.551,Z 476.03,A -85,B 0,C 180,E1 761.824,E2 761.824} C_VEL
LIN {X 0,Y 609.723,Z 476.03,A -85,B 0,C 180,E1 766.066,E2 766.066} C_VEL
LIN {X 0,Y 609.539,Z 476.03,A -85,B 0,C 180,E1 770.357,E2 770.357} C_VEL
LIN {X 0,Y 609.571,Z 476.03,A -85,B 0,C 180,E1 775.159,E2 775.159} C_VEL
LIN {X 0,Y 609.745,Z 476.03,A -85,B 0,C 180,E1 780.353,E2 780.353} C_VEL
LIN {X 0,Y 609.99,Z 476.03,A -85,B 0,C 180,E1 785.041,E2 785.041} C_VEL
LIN {X 0,Y 609.795,Z 476.03,A -85,B 0,C 180,E1 791.169,E2 791.169} C_VEL
LIN {X 0,Y 609.715,Z 476.03,A -85,B 0,C 180,E1 797.086,E2 797.086} C_VEL
LIN {X 0,Y 610.04,Z 476.03,A -85,B 0,C 180,E1 798.548,E2 798.548} C_VEL
LIN {X 0,Y 610.684,Z 519.008,A -85,B 0,C 180,E1 799.915,E2 799.915} C_VEL
LIN {X 0,Y 610.558,Z 557.222,A -85,B 0,C 180,E1 801.739,E2 801.739} C_VEL
LIN {X 0,Y 610.408,Z 591.799,A -85,B 0,C 180,E1 804.011,E2 804.011} C_VEL
LIN {X 0,Y 610.287,Z 622.15,A -85,B 0,C 180,E1 806.622,E2 806.622} C_VEL
LIN {X 0,Y 610.159,Z 649.335,A -85,B 0,C 180,E1 809.645,E2 809.645} C_VEL
LIN {X 0,Y 610.12,Z 672.481,A -85,B 0,C 180,E1 813.023,E2 813.023} C_VEL
LIN {X 0,Y 610.133,Z 689.91,A -85,B 0,C 180,E1 816.484,E2 816.484} C_VEL
LIN {X 0,Y 610.099,Z 702.09,A -85,B 0,C 180,E1 820.005,E2 820.005} C_VEL
LIN {X 0,Y 610.006,Z 708.309,A -85,B 0,C 180,E1 822.909,E2 822.909} C_VEL
LIN {X 0,Y 609.913,Z 711.246,A -85,B 0,C 180,E1 825.848,E2 825.848} C_VEL
LIN {X 0,Y 610.085,Z 710.328,A -85,B 0,C 180,E1 829.429,E2 829.429} C_VEL
LIN {X 0,Y 609.986,Z 703.698,A -85,B 0,C 180,E1 833.308,E2 833.308} C_VEL
LIN {X 0,Y 610.005,Z 691.858,A -85,B 0,C 180,E1 836.972,E2 836.972} C_VEL
LIN {X 0,Y 610.087,Z 674.31,A -85,B 0,C 180,E1 840.582,E2 840.582} C_VEL
LIN {X 0,Y 610.173,Z 651.897,A -85,B 0,C 180,E1 843.941,E2 843.941} C_VEL
LIN {X 0,Y 610.275,Z 624.029,A -85,B 0,C 180,E1 847.103,E2 847.103} C_VEL
LIN {X 0,Y 610.359,Z 593.937,A -85,B 0,C 180,E1 849.736,E2 849.736} C_VEL
LIN {X 0,Y 610.547,Z 559.554,A -85,B 0,C 180,E1 852.035,E2 852.035} C_VEL
LIN {X 0,Y 610.612,Z 522.609,A -85,B 0,C 180,E1 853.849,E2 853.849} C_VEL
LIN {X 0,Y 610.635,Z 483.876,A -85,B 0,C 180,E1 855.13,E2 855.13} C_VEL
LIN {X 0,Y 609.959,Z 476.03,A -85,B 0,C 180,E1 855.411,E2 855.411} C_VEL
LIN {X 0,Y 609.769,Z 476.03,A -85,B 0,C 180,E1 861.628,E2 861.628} C_VEL
LIN {X 0,Y 609.787,Z 476.03,A -85,B 0,C 180,E1 867.59,E2 867.59} C_VEL
LIN {X 0,Y 609.969,Z 476.03,A -85,B 0,C 180,E1 871.859,E2 871.859} C_VEL
LIN {X 0,Y 609.757,Z 476.03,A -85,B 0,C 180,E1 878.131,E2 878.131} C_VEL
LIN {X 0,Y 610.039,Z 476.03,A -85,B 0,C 180,E1 882.671,E2 882.671} C_VEL
LIN {X 0,Y 608.654,Z 476.03,A -85,B 0,C 180,E1 882.957,E2 882.957} C_VEL
LIN {X 0,Y 610.423,Z 489.354,A -85,B 0,C 180,E1 883.24,E2 883.24} C_VEL
LIN {X 0,Y 610.348,Z 521.111,A -85,B 0,C 180,E1 884.206,E2 884.206} C_VEL
LIN {X 0,Y 610.31,Z 550.569,A -85,B 0,C 180,E1 885.726,E2 885.726} C_VEL
LIN {X 0,Y 610.244,Z 575.626,A -85,B 0,C 180,E1 887.642,E2 887.642} C_VEL
LIN {X 0,Y 610.201,Z 597.179,A -85,B 0,C 180,E1 889.996,E2 889.996} C_VEL
LIN {X 0,Y 610.139,Z 613.634,A -85,B 0,C 180,E1 892.606,E2 892.606} C_VEL
LIN {X 0,Y 610.136,Z 619.876,A -85,B 0,C 180,E1 893.98,E2 893.98} C_VEL
LIN {X 0,Y 607.602,Z 624.072,A -85,B 0,C 180,E1 895.131,E2 895.131} C_VEL
LIN {X 0,Y 602.304,Z 628.587,A -85,B 0,C 180,E1 896.89,E2 896.89} C_VEL
LIN {X 0,Y 602.234,Z 628.938,A -85,B 0,C 180,E1 897.095,E2 897.095} C_VEL
LIN {X 0,Y 602.211,Z 631.497,A -85,B 0,C 180,E1 899.998,E2 899.998} C_VEL
LIN {X 0,Y 602.217,Z 628.838,A -85,B 0,C 180,E1 902.88,E2 902.88} C_VEL
LIN {X 0,Y 602.242,Z 620.782,A -85,B 0,C 180,E1 905.769,E2 905.769} C_VEL
LIN {X 0,Y 602.293,Z 606.526,A -85,B 0,C 180,E1 908.672,E2 908.672} C_VEL
LIN {X 0,Y 602.382,Z 587.312,A -85,B 0,C 180,E1 911.244,E2 911.244} C_VEL
LIN {X 0,Y 602.523,Z 563.732,A -85,B 0,C 180,E1 913.438,E2 913.438} C_VEL
LIN {X 0,Y 602.687,Z 535.596,A -85,B 0,C 180,E1 915.235,E2 915.235} C_VEL
LIN {X 0,Y 602.819,Z 505.096,A -85,B 0,C 180,E1 916.478,E2 916.478} C_VEL
LIN {X 0,Y 602.134,Z 476.03,A -85,B 0,C 180,E1 917.148,E2 917.148} C_VEL
LIN {X 0,Y 601.65,Z 476.03,A -85,B 0,C 180,E1 922.174,E2 922.174} C_VEL
LIN {X 0,Y 601.975,Z 476.03,A -85,B 0,C 180,E1 925.31,E2 925.31} C_VEL
LIN {X 0,Y 601.681,Z 476.03,A -85,B 0,C 180,E1 931.173,E2 931.173} C_VEL
LIN {X 0,Y 601.759,Z 476.03,A -85,B 0,C 180,E1 937.142,E2 937.142} C_VEL
LIN {X 0,Y 601.777,Z 476.03,A -85,B 0,C 180,E1 943.142,E2 943.142} C_VEL
LIN {X 0,Y 601.583,Z 476.03,A -85,B 0,C 180,E1 949.126,E2 949.126} C_VEL
LIN {X 0,Y 601.5,Z 476.03,A -85,B 0,C 180,E1 953.651,E2 953.651} C_VEL
LIN {X 0,Y 601.937,Z 476.03,A -85,B 0,C 180,E1 958.113,E2 958.113} C_VEL
LIN {X 0,Y 602.059,Z 476.03,A -85,B 0,C 180,E1 960.12,E2 960.12} C_VEL
LIN {X 0,Y 603.334,Z 486.104,A -85,B 0,C 180,E1 960.337,E2 960.337} C_VEL
LIN {X 0,Y 603.772,Z 547.156,A -85,B 0,C 180,E1 961.305,E2 961.305} C_VEL
LIN {X 0,Y 603.642,Z 587.087,A -85,B 0,C 180,E1 962.539,E2 962.539} C_VEL
LIN {X 0,Y 603.312,Z 625.325,A -85,B 0,C 180,E1 964.348,E2 964.348} C_VEL
LIN {X 0,Y 602.968,Z 661.359,A -85,B 0,C 180,E1 966.722,E2 966.722} C_VEL
LIN {X 0,Y 602.659,Z 693.292,A -85,B 0,C 180,E1 969.512,E2 969.512} C_VEL
LIN {X 0,Y 602.43,Z 720.87,A -85,B 0,C 180,E1 972.657,E2 972.657} C_VEL
LIN {X 0,Y 602.29,Z 744.253,A -85,B 0,C 180,E1 976.183,E2 976.183} C_VEL
LIN {X 0,Y 602.246,Z 761.905,A -85,B 0,C 180,E1 979.864,E2 979.864} C_VEL
LIN {X 0,Y 602.178,Z 774.115,A -85,B 0,C 180,E1 983.733,E2 983.733} C_VEL
LIN {X 0,Y 602.114,Z 779.897,A -85,B 0,C 180,E1 987.117,E2 987.117} C_VEL
LIN {X 0,Y 602.077,Z 781.5,A -85,B 0,C 180,E1 990,E2 990} C_VEL
LIN {X 0,Y 602.197,Z 779.897,A -85,B 0,C 180,E1 992.882,E2 992.882} C_VEL
LIN {X 0,Y 602.135,Z 772.88,A -85,B 0,C 180,E1 996.746,E2 996.746} C_VEL
LIN {X 0,Y 602.208,Z 760.618,A -85,B 0,C 180,E1 1000.444,E2 1000.444} C_VEL
LIN {X 0,Y 602.235,Z 743.16,A -85,B 0,C 180,E1 1004.004,E2 1004.004} C_VEL
LIN {X 0,Y 602.4,Z 720.963,A -85,B 0,C 180,E1 1007.332,E2 1007.332} C_VEL
LIN {X 0,Y 602.645,Z 693.315,A -85,B 0,C 180,E1 1010.486,E2 1010.486} C_VEL
LIN {X 0,Y 602.96,Z 661.394,A -85,B 0,C 180,E1 1013.276,E2 1013.276} C_VEL
LIN {X 0,Y 603.259,Z 625.335,A -85,B 0,C 180,E1 1015.654,E2 1015.654} C_VEL
LIN {X 0,Y 603.488,Z 585.495,A -85,B 0,C 180,E1 1017.529,E2 1017.529} C_VEL
LIN {X 0,Y 603.871,Z 545.728,A -85,B 0,C 180,E1 1018.722,E2 1018.722} C_VEL
LIN {X 0,Y 602.815,Z 479.02,A -85,B 0,C 180,E1 1019.787,E2 1019.787} C_VEL
LIN {X 0,Y 602.203,Z 476.03,A -85,B 0,C 180,E1 1019.908,E2 1019.908} C_VEL
LIN {X 0,Y 601.73,Z 476.03,A -85,B 0,C 180,E1 1027.15,E2 1027.15} C_VEL
LIN {X 0,Y 601.749,Z 476.03,A -85,B 0,C 180,E1 1033.147,E2 1033.147} C_VEL
LIN {X 0,Y 601.568,Z 476.03,A -85,B 0,C 180,E1 1039.132,E2 1039.132} C_VEL
LIN {X 0,Y 601.501,Z 476.03,A -85,B 0,C 180,E1 1043.659,E2 1043.659} C_VEL
LIN {X 0,Y 601.812,Z 476.03,A -85,B 0,C 180,E1 1048.112,E2 1048.112} C_VEL
LIN {X 0,Y 601.646,Z 476.03,A -85,B 0,C 180,E1 1053.069,E2 1053.069} C_VEL
LIN {X 0,Y 601.664,Z 476.03,A -85,B 0,C 180,E1 1058.61,E2 1058.61} C_VEL
LIN {X 0,Y 602.027,Z 476.03,A -85,B 0,C 180,E1 1062.883,E2 1062.883} C_VEL
LIN {X 0,Y 601.835,Z 476.03,A -85,B 0,C 180,E1 1068.392,E2 1068.392} C_VEL
LIN {X 0,Y 601.876,Z 476.03,A -85,B 0,C 180,E1 1072.777,E2 1072.777} C_VEL
LIN {X 0,Y 602.034,Z 476.03,A -85,B 0,C 180,E1 1077.119,E2 1077.119} C_VEL
LIN {X 0,Y 602.137,Z 476.03,A -85,B 0,C 180,E1 1081.443,E2 1081.443} C_VEL
LIN {X 0,Y 602.194,Z 476.03,A -85,B 0,C 180,E1 1085.774,E2 1085.774} C_VEL
LIN {X 0,Y 601.834,Z 476.03,A -85,B 0,C 180,E1 1091.612,E2 1091.612} C_VEL
LIN {X 0,Y 601.681,Z 476.03,A -85,B 0,C 180,E1 1097.009,E2 1097.009} C_VEL
LIN {X 0,Y 601.665,Z 476.03,A -85,B 0,C 180,E1 1102.178,E2 1102.178} C_VEL
LIN {X 0,Y 601.987,Z 476.03,A -85,B 0,C 180,E1 1105.315,E2 1105.315} C_VEL
LIN {X 0,Y 601.743,Z 476.03,A -85,B 0,C 180,E1 1111.184,E2 1111.184} C_VEL
LIN {X 0,Y 601.889,Z 476.03,A -85,B 0,C 180,E1 1117.138,E2 1117.138} C_VEL
LIN {X 0,Y 601.62,Z 476.03,A -85,B 0,C 180,E1 1123.126,E2 1123.126} C_VEL
LIN {X 0,Y 601.804,Z 476.03,A -85,B 0,C 180,E1 1127.211,E2 1127.211} C_VEL
LIN {X 0,Y 601.753,Z 476.03,A -85,B 0,C 180,E1 1132.852,E2 1132.852} C_VEL
LIN {X 0,Y 601.698,Z 476.03,A -85,B 0,C 180,E1 1138.821,E2 1138.821} C_VEL
LIN {X 0,Y 602.036,Z 476.03,A -85,B 0,C 180,E1 1144.873,E2 1144.873} C_VEL
LIN {X 0,Y 601.935,Z 476.03,A -85,B 0,C 180,E1 1150.913,E2 1150.913} C_VEL
LIN {X 0,Y 601.784,Z 476.03,A -85,B 0,C 180,E1 1156.912,E2 1156.912} C_VEL
LIN {X 0,Y 602.025,Z 476.03,A -85,B 0,C 180,E1 1158.129,E2 1158.129} C_VEL
LIN {X 0,Y 603.636,Z 485.562,A -85,B 0,C 180,E1 1158.467,E2 1158.467} C_VEL
LIN {X 0,Y 603.513,Z 524.415,A -85,B 0,C 180,E1 1159.794,E2 1159.794} C_VEL
LIN {X 0,Y 603.229,Z 560.614,A -85,B 0,C 180,E1 1161.611,E2 1161.611} C_VEL
LIN {X 0,Y 602.901,Z 595.414,A -85,B 0,C 180,E1 1163.991,E2 1163.991} C_VEL
LIN {X 0,Y 602.621,Z 626.223,A -85,B 0,C 180,E1 1166.759,E2 1166.759} C_VEL
LIN {X 0,Y 602.434,Z 653.829,A -85,B 0,C 180,E1 1170,E2 1170} C_VEL
LIN {X 0,Y 602.306,Z 674.854,A -85,B 0,C 180,E1 1173.243,E2 1173.243} C_VEL
LIN {X 0,Y 602.261,Z 691.838,A -85,B 0,C 180,E1 1176.802,E2 1176.802} C_VEL
LIN {X 0,Y 602.238,Z 704.16,A -85,B 0,C 180,E1 1180.709,E2 1180.709} C_VEL
LIN {X 0,Y 602.137,Z 710.417,A -85,B 0,C 180,E1 1184.564,E2 1184.564} C_VEL
LIN {X 0,Y 602.144,Z 711.366,A -85,B 0,C 180,E1 1187.563,E2 1187.563} C_VEL
LIN {X 0,Y 602.094,Z 707.574,A -85,B 0,C 180,E1 1191.499,E2 1191.499} C_VEL
LIN {X 0,Y 602.152,Z 698.729,A -85,B 0,C 180,E1 1195.151,E2 1195.151} C_VEL
LIN {X 0,Y 602.219,Z 685.688,A -85,B 0,C 180,E1 1198.536,E2 1198.536} C_VEL
LIN {X 0,Y 602.314,Z 666.18,A -85,B 0,C 180,E1 1202.109,E2 1202.109} C_VEL
LIN {X 0,Y 602.492,Z 641.758,A -85,B 0,C 180,E1 1205.432,E2 1205.432} C_VEL
LIN {X 0,Y 602.738,Z 612.926,A -85,B 0,C 180,E1 1208.433,E2 1208.433} C_VEL
LIN {X 0,Y 603.033,Z 580.87,A -85,B 0,C 180,E1 1210.999,E2 1210.999} C_VEL
LIN {X 0,Y 603.358,Z 545.381,A -85,B 0,C 180,E1 1213.14,E2 1213.14} C_VEL
LIN {X 0,Y 603.694,Z 507.161,A -85,B 0,C 180,E1 1214.778,E2 1214.778} C_VEL
LIN {X 0,Y 602.784,Z 479.492,A -85,B 0,C 180,E1 1215.644,E2 1215.644} C_VEL
LIN {X 0,Y 601.935,Z 476.03,A -85,B 0,C 180,E1 1215.81,E2 1215.81} C_VEL
LIN {X 0,Y 601.779,Z 476.03,A -85,B 0,C 180,E1 1221.259,E2 1221.259} C_VEL
LIN {X 0,Y 601.908,Z 476.03,A -85,B 0,C 180,E1 1226.398,E2 1226.398} C_VEL
LIN {X 0,Y 602.02,Z 476.03,A -85,B 0,C 180,E1 1231.676,E2 1231.676} C_VEL
LIN {X 0,Y 601.838,Z 476.03,A -85,B 0,C 180,E1 1237.828,E2 1237.828} C_VEL
LIN {X 0,Y 601.522,Z 476.03,A -85,B 0,C 180,E1 1242.625,E2 1242.625} C_VEL
LIN {X 0,Y 601.094,Z 477.394,A -85,B 0,C 180,E1 1242.763,E2 1242.763} C_VEL
LIN {X 0,Y 602.842,Z 491.707,A -85,B 0,C 180,E1 1243.077,E2 1243.077} C_VEL
LIN {X 0,Y 602.714,Z 522.272,A -85,B 0,C 180,E1 1244.051,E2 1244.051} C_VEL
LIN {X 0,Y 602.594,Z 550.558,A -85,B 0,C 180,E1 1245.539,E2 1245.539} C_VEL
LIN {X 0,Y 602.476,Z 575.615,A -85,B 0,C 180,E1 1247.48,E2 1247.48} C_VEL
LIN {X 0,Y 602.356,Z 597.178,A -85,B 0,C 180,E1 1249.864,E2 1249.864} C_VEL
LIN {X 0,Y 602.269,Z 613.157,A -85,B 0,C 180,E1 1252.414,E2 1252.414} C_VEL
LIN {X 0,Y 602.256,Z 624.74,A -85,B 0,C 180,E1 1255.311,E2 1255.311} C_VEL
LIN {X 0,Y 602.234,Z 628.938,A -85,B 0,C 180,E1 1257.095,E2 1257.095} C_VEL
LIN {X 0,Y 599.783,Z 630.799,A -85,B 0,C 180,E1 1258.307,E2 1258.307} C_VEL
LIN {X 0,Y 594.381,Z 631.469,A -85,B 0,C 180,E1 1260.138,E2 1260.138} C_VEL
LIN {X 0,Y 594.273,Z 631.333,A -85,B 0,C 180,E1 1260.35,E2 1260.35} C_VEL
LIN {X 0,Y 594.318,Z 628.839,A -85,B 0,C 180,E1 1262.918,E2 1262.918} C_VEL
LIN {X 0,Y 594.353,Z 620.789,A -85,B 0,C 180,E1 1265.846,E2 1265.846} C_VEL
LIN {X 0,Y 594.428,Z 606.534,A -85,B 0,C 180,E1 1268.788,E2 1268.788} C_VEL
LIN {X 0,Y 594.578,Z 587.323,A -85,B 0,C 180,E1 1271.393,E2 1271.393} C_VEL
LIN {X 0,Y 594.776,Z 563.773,A -85,B 0,C 180,E1 1273.614,E2 1273.614} C_VEL
LIN {X 0,Y 595.013,Z 536.334,A -85,B 0,C 180,E1 1275.399,E2 1275.399} C_VEL
LIN {X 0,Y 595.239,Z 506.191,A -85,B 0,C 180,E1 1276.662,E2 1276.662} C_VEL
LIN {X 0,Y 594.562,Z 478.368,A -85,B 0,C 180,E1 1277.328,E2 1277.328} C_VEL
LIN {X 0,Y 594.183,Z 476.03,A -85,B 0,C 180,E1 1277.385,E2 1277.385} C_VEL
LIN {X 0,Y 593.732,Z 476.03,A -85,B 0,C 180,E1 1282.486,E2 1282.486} C_VEL
LIN {X 0,Y 593.72,Z 476.03,A -85,B 0,C 180,E1 1287.32,E2 1287.32} C_VEL
LIN {X 0,Y 593.602,Z 476.03,A -85,B 0,C 180,E1 1292.383,E2 1292.383} C_VEL
LIN {X 0,Y 593.801,Z 476.03,A -85,B 0,C 180,E1 1297.771,E2 1297.771} C_VEL
LIN {X 0,Y 593.832,Z 476.03,A -85,B 0,C 180,E1 1303.499,E2 1303.499} C_VEL
LIN {X 0,Y 593.636,Z 476.03,A -85,B 0,C 180,E1 1308.459,E2 1308.459} C_VEL
LIN {X 0,Y 593.635,Z 476.03,A -85,B 0,C 180,E1 1314.081,E2 1314.081} C_VEL
LIN {X 0,Y 594.065,Z 476.03,A -85,B 0,C 180,E1 1319.667,E2 1319.667} C_VEL
LIN {X 0,Y 596.459,Z 485.177,A -85,B 0,C 180,E1 1319.947,E2 1319.947} C_VEL
LIN {X 0,Y 596.824,Z 547.883,A -85,B 0,C 180,E1 1320.956,E2 1320.956} C_VEL
LIN {X 0,Y 596.567,Z 587.486,A -85,B 0,C 180,E1 1322.202,E2 1322.202} C_VEL
LIN {X 0,Y 596.029,Z 625.308,A -85,B 0,C 180,E1 1324.01,E2 1324.01} C_VEL
LIN {X 0,Y 595.499,Z 661.302,A -85,B 0,C 180,E1 1326.407,E2 1326.407} C_VEL
LIN {X 0,Y 595.026,Z 692.237,A -85,B 0,C 180,E1 1329.13,E2 1329.13} C_VEL
LIN {X 0,Y 594.671,Z 719.231,A -85,B 0,C 180,E1 1332.209,E2 1332.209} C_VEL
LIN {X 0,Y 594.464,Z 740.848,A -85,B 0,C 180,E1 1335.411,E2 1335.411} C_VEL
LIN {X 0,Y 594.291,Z 758.678,A -85,B 0,C 180,E1 1338.948,E2 1338.948} C_VEL
LIN {X 0,Y 594.232,Z 771.619,A -85,B 0,C 180,E1 1342.68,E2 1342.68} C_VEL
LIN {X 0,Y 594.154,Z 777.936,A -85,B 0,C 180,E1 1345.615,E2 1345.615} C_VEL
LIN {X 0,Y 594.164,Z 781.086,A -85,B 0,C 180,E1 1348.54,E2 1348.54} C_VEL
LIN {X 0,Y 594.337,Z 781.086,A -85,B 0,C 180,E1 1351.46,E2 1351.46} C_VEL
LIN {X 0,Y 594.141,Z 776.724,A -85,B 0,C 180,E1 1355.117,E2 1355.117} C_VEL
LIN {X 0,Y 594.223,Z 767.214,A -85,B 0,C 180,E1 1358.794,E2 1358.794} C_VEL
LIN {X 0,Y 594.265,Z 752.083,A -85,B 0,C 180,E1 1362.507,E2 1362.507} C_VEL
LIN {X 0,Y 594.466,Z 731.564,A -85,B 0,C 180,E1 1366.08,E2 1366.08} C_VEL
LIN {X 0,Y 594.824,Z 704.954,A -85,B 0,C 180,E1 1369.524,E2 1369.524} C_VEL
LIN {X 0,Y 595.277,Z 675.531,A -85,B 0,C 180,E1 1372.428,E2 1372.428} C_VEL
LIN {X 0,Y 595.789,Z 642.385,A -85,B 0,C 180,E1 1374.939,E2 1374.939} C_VEL
LIN {X 0,Y 596.302,Z 607.177,A -85,B 0,C 180,E1 1376.933,E2 1376.933} C_VEL
LIN {X 0,Y 596.69,Z 571.159,A -85,B 0,C 180,E1 1378.385,E2 1378.385} C_VEL
LIN {X 0,Y 597.119,Z 533.455,A -85,B 0,C 180,E1 1379.332,E2 1379.332} C_VEL
LIN {X 0,Y 595.807,Z 480.835,A -85,B 0,C 180,E1 1380.148,E2 1380.148} C_VEL
LIN {X 0,Y 594.116,Z 476.03,A -85,B 0,C 180,E1 1380.342,E2 1380.342} C_VEL
LIN {X 0,Y 593.838,Z 476.03,A -85,B 0,C 180,E1 1385.904,E2 1385.904} C_VEL
LIN {X 0,Y 593.786,Z 476.03,A -85,B 0,C 180,E1 1391.527,E2 1391.527} C_VEL
LIN {X 0,Y 593.69,Z 476.03,A -85,B 0,C 180,E1 1396.488,E2 1396.488} C_VEL
LIN {X 0,Y 593.716,Z 476.03,A -85,B 0,C 180,E1 1402.268,E2 1402.268} C_VEL
LIN {X 0,Y 593.886,Z 476.03,A -85,B 0,C 180,E1 1407.635,E2 1407.635} C_VEL
LIN {X 0,Y 593.734,Z 476.03,A -85,B 0,C 180,E1 1413.196,E2 1413.196} C_VEL
LIN {X 0,Y 593.778,Z 476.03,A -85,B 0,C 180,E1 1417.516,E2 1417.516} C_VEL
LIN {X 0,Y 594.063,Z 476.03,A -85,B 0,C 180,E1 1422.194,E2 1422.194} C_VEL
LIN {X 0,Y 593.944,Z 476.03,A -85,B 0,C 180,E1 1428.236,E2 1428.236} C_VEL
LIN {X 0,Y 593.987,Z 476.03,A -85,B 0,C 180,E1 1432.68,E2 1432.68} C_VEL
LIN {X 0,Y 594.127,Z 476.03,A -85,B 0,C 180,E1 1437.081,E2 1437.081} C_VEL
LIN {X 0,Y 594.226,Z 476.03,A -85,B 0,C 180,E1 1441.462,E2 1441.462} C_VEL
LIN {X 0,Y 594.096,Z 476.03,A -85,B 0,C 180,E1 1446.305,E2 1446.305} C_VEL
LIN {X 0,Y 593.896,Z 476.03,A -85,B 0,C 180,E1 1451.77,E2 1451.77} C_VEL
LIN {X 0,Y 593.896,Z 476.03,A -85,B 0,C 180,E1 1456.288,E2 1456.288} C_VEL
LIN {X 0,Y 593.974,Z 476.03,A -85,B 0,C 180,E1 1460.909,E2 1460.909} C_VEL
LIN {X 0,Y 593.969,Z 476.03,A -85,B 0,C 180,E1 1465.681,E2 1465.681} C_VEL
LIN {X 0,Y 593.884,Z 476.03,A -85,B 0,C 180,E1 1470.657,E2 1470.657} C_VEL
LIN {X 0,Y 593.884,Z 476.03,A -85,B 0,C 180,E1 1475.901,E2 1475.901} C_VEL
LIN {X 0,Y 593.644,Z 476.03,A -85,B 0,C 180,E1 1481.539,E2 1481.539} C_VEL
LIN {X 0,Y 593.836,Z 476.03,A -85,B 0,C 180,E1 1486.495,E2 1486.495} C_VEL
LIN {X 0,Y 593.792,Z 476.03,A -85,B 0,C 180,E1 1492.268,E2 1492.268} C_VEL
LIN {X 0,Y 593.609,Z 476.03,A -85,B 0,C 180,E1 1497.613,E2 1497.613} C_VEL
LIN {X 0,Y 593.718,Z 476.03,A -85,B 0,C 180,E1 1502.675,E2 1502.675} C_VEL
LIN {X 0,Y 593.727,Z 476.03,A -85,B 0,C 180,E1 1507.51,E2 1507.51} C_VEL
LIN {X 0,Y 593.951,Z 476.03,A -85,B 0,C 180,E1 1512.188,E2 1512.188} C_VEL
LIN {X 0,Y 594.022,Z 476.152,A -85,B 0,C 180,E1 1517.721,E2 1517.721} C_VEL
LIN {X 0,Y 596.677,Z 486.584,A -85,B 0,C 180,E1 1518.131,E2 1518.131} C_VEL
LIN {X 0,Y 596.37,Z 525.301,A -85,B 0,C 180,E1 1519.48,E2 1519.48} C_VEL
LIN {X 0,Y 595.948,Z 561.37,A -85,B 0,C 180,E1 1521.324,E2 1521.324} C_VEL
LIN {X 0,Y 595.417,Z 595.65,A -85,B 0,C 180,E1 1523.704,E2 1523.704} C_VEL
LIN {X 0,Y 594.996,Z 626.682,A -85,B 0,C 180,E1 1526.535,E2 1526.535} C_VEL
LIN {X 0,Y 594.64,Z 654.157,A -85,B 0,C 180,E1 1529.818,E2 1529.818} C_VEL
LIN {X 0,Y 594.46,Z 676.072,A -85,B 0,C 180,E1 1533.286,E2 1533.286} C_VEL
LIN {X 0,Y 594.395,Z 692.407,A -85,B 0,C 180,E1 1536.816,E2 1536.816} C_VEL
LIN {X 0,Y 594.341,Z 704.516,A -85,B 0,C 180,E1 1540.792,E2 1540.792} C_VEL
LIN {X 0,Y 594.22,Z 710.578,A -85,B 0,C 180,E1 1544.762,E2 1544.762} C_VEL
LIN {X 0,Y 594.219,Z 711.312,A -85,B 0,C 180,E1 1547.805,E2 1547.805} C_VEL
LIN {X 0,Y 594.242,Z 708.658,A -85,B 0,C 180,E1 1550.899,E2 1550.899} C_VEL
LIN {X 0,Y 594.322,Z 700.335,A -85,B 0,C 180,E1 1554.744,E2 1554.744} C_VEL
LIN {X 0,Y 594.362,Z 686.703,A -85,B 0,C 180,E1 1558.474,E2 1558.474} C_VEL
LIN {X 0,Y 594.494,Z 667.131,A -85,B 0,C 180,E1 1562.165,E2 1562.165} C_VEL
LIN {X 0,Y 594.769,Z 642.425,A -85,B 0,C 180,E1 1565.601,E2 1565.601} C_VEL
LIN {X 0,Y 595.171,Z 613.85,A -85,B 0,C 180,E1 1568.633,E2 1568.633} C_VEL
LIN {X 0,Y 595.636,Z 581.215,A -85,B 0,C 180,E1 1571.293,E2 1571.293} C_VEL
LIN {X 0,Y 596.153,Z 545.386,A -85,B 0,C 180,E1 1573.481,E2 1573.481} C_VEL
LIN {X 0,Y 596.64,Z 507.256,A -85,B 0,C 180,E1 1575.132,E2 1575.132} C_VEL
LIN {X 0,Y 595.898,Z 482.291,A -85,B 0,C 180,E1 1575.934,E2 1575.934} C_VEL
LIN {X 0,Y 593.884,Z 476.03,A -85,B 0,C 180,E1 1576.255,E2 1576.255} C_VEL
LIN {X 0,Y 593.703,Z 476.03,A -85,B 0,C 180,E1 1582.261,E2 1582.261} C_VEL
LIN {X 0,Y 593.873,Z 476.03,A -85,B 0,C 180,E1 1587.628,E2 1587.628} C_VEL
LIN {X 0,Y 593.835,Z 476.03,A -85,B 0,C 180,E1 1592.68,E2 1592.68} C_VEL
LIN {X 0,Y 593.88,Z 476.03,A -85,B 0,C 180,E1 1597.515,E2 1597.515} C_VEL
LIN {X 0,Y 593.593,Z 476.03,A -85,B 0,C 180,E1 1602.506,E2 1602.506} C_VEL
LIN {X 0,Y 595.27,Z 496.021,A -85,B 0,C 180,E1 1602.959,E2 1602.959} C_VEL
LIN {X 0,Y 595.062,Z 526.504,A -85,B 0,C 180,E1 1604.03,E2 1604.03} C_VEL
LIN {X 0,Y 594.833,Z 554.968,A -85,B 0,C 180,E1 1605.647,E2 1605.647} C_VEL
LIN {X 0,Y 594.652,Z 579.459,A -85,B 0,C 180,E1 1607.686,E2 1607.686} C_VEL
LIN {X 0,Y 594.482,Z 599.844,A -85,B 0,C 180,E1 1610.099,E2 1610.099} C_VEL
LIN {X 0,Y 594.378,Z 614.92,A -85,B 0,C 180,E1 1612.681,E2 1612.681} C_VEL
LIN {X 0,Y 594.334,Z 625.739,A -85,B 0,C 180,E1 1615.615,E2 1615.615} C_VEL
LIN {X 0,Y 594.3,Z 630.887,A -85,B 0,C 180,E1 1618.538,E2 1618.538} C_VEL
LIN {X 0,Y 594.273,Z 631.333,A -85,B 0,C 180,E1 1620.35,E2 1620.35} C_VEL
LIN {X 0,Y 591.719,Z 630.697,A -85,B 0,C 180,E1 1621.587,E2 1621.587} C_VEL
LIN {X 0,Y 586.534,Z 627.921,A -85,B 0,C 180,E1 1623.425,E2 1623.425} C_VEL
LIN {X 0,Y 586.469,Z 627.476,A -85,B 0,C 180,E1 1623.635,E2 1623.635} C_VEL
LIN {X 0,Y 586.491,Z 618.044,A -85,B 0,C 180,E1 1626.624,E2 1626.624} C_VEL
LIN {X 0,Y 586.629,Z 603.032,A -85,B 0,C 180,E1 1629.468,E2 1629.468} C_VEL
LIN {X 0,Y 586.849,Z 582.302,A -85,B 0,C 180,E1 1632.098,E2 1632.098} C_VEL
LIN {X 0,Y 587.113,Z 557.849,A -85,B 0,C 180,E1 1634.25,E2 1634.25} C_VEL
LIN {X 0,Y 587.431,Z 530.75,A -85,B 0,C 180,E1 1635.891,E2 1635.891} C_VEL
LIN {X 0,Y 587.688,Z 500.856,A -85,B 0,C 180,E1 1637.043,E2 1637.043} C_VEL
LIN {X 0,Y 587.071,Z 479.876,A -85,B 0,C 180,E1 1637.534,E2 1637.534} C_VEL
LIN {X 0,Y 586.259,Z 476.03,A -85,B 0,C 180,E1 1637.665,E2 1637.665} C_VEL
LIN {X 0,Y 585.865,Z 476.03,A -85,B 0,C 180,E1 1642.805,E2 1642.805} C_VEL
LIN {X 0,Y 585.776,Z 476.03,A -85,B 0,C 180,E1 1647.723,E2 1647.723} C_VEL
LIN {X 0,Y 585.7,Z 476.03,A -85,B 0,C 180,E1 1652.874,E2 1652.874} C_VEL
LIN {X 0,Y 585.841,Z 476.03,A -85,B 0,C 180,E1 1658.331,E2 1658.331} C_VEL
LIN {X 0,Y 585.917,Z 476.03,A -85,B 0,C 180,E1 1664.238,E2 1664.238} C_VEL
LIN {X 0,Y 585.797,Z 476.03,A -85,B 0,C 180,E1 1669.746,E2 1669.746} C_VEL
LIN {X 0,Y 586.009,Z 476.03,A -85,B 0,C 180,E1 1675.762,E2 1675.762} C_VEL
LIN {X 0,Y 586.127,Z 476.03,A -85,B 0,C 180,E1 1679.222,E2 1679.222} C_VEL
LIN {X 0,Y 589.631,Z 485.399,A -85,B 0,C 180,E1 1679.566,E2 1679.566} C_VEL
LIN {X 0,Y 589.909,Z 547.688,A -85,B 0,C 180,E1 1680.578,E2 1680.578} C_VEL
LIN {X 0,Y 589.51,Z 587.458,A -85,B 0,C 180,E1 1681.839,E2 1681.839} C_VEL
LIN {X 0,Y 588.821,Z 624.16,A -85,B 0,C 180,E1 1683.601,E2 1683.601} C_VEL
LIN {X 0,Y 588.11,Z 660.005,A -85,B 0,C 180,E1 1685.988,E2 1685.988} C_VEL
LIN {X 0,Y 587.461,Z 692.241,A -85,B 0,C 180,E1 1688.848,E2 1688.848} C_VEL
LIN {X 0,Y 586.927,Z 719.236,A -85,B 0,C 180,E1 1691.966,E2 1691.966} C_VEL
LIN {X 0,Y 586.627,Z 741.628,A -85,B 0,C 180,E1 1695.348,E2 1695.348} C_VEL
LIN {X 0,Y 586.42,Z 758.788,A -85,B 0,C 180,E1 1698.824,E2 1698.824} C_VEL
LIN {X 0,Y 586.335,Z 771.622,A -85,B 0,C 180,E1 1702.581,E2 1702.581} C_VEL
LIN {X 0,Y 586.251,Z 777.939,A -85,B 0,C 180,E1 1705.556,E2 1705.556} C_VEL
LIN {X 0,Y 586.271,Z 781.088,A -85,B 0,C 180,E1 1708.52,E2 1708.52} C_VEL
LIN {X 0,Y 586.434,Z 781.089,A -85,B 0,C 180,E1 1711.479,E2 1711.479} C_VEL
LIN {X 0,Y 586.266,Z 776.723,A -85,B 0,C 180,E1 1715.186,E2 1715.186} C_VEL
LIN {X 0,Y 586.334,Z 767.217,A -85,B 0,C 180,E1 1718.913,E2 1718.913} C_VEL
LIN {X 0,Y 586.428,Z 752.086,A -85,B 0,C 180,E1 1722.677,E2 1722.677} C_VEL
LIN {X 0,Y 586.669,Z 731.567,A -85,B 0,C 180,E1 1726.3,E2 1726.3} C_VEL
LIN {X 0,Y 587.191,Z 705.183,A -85,B 0,C 180,E1 1729.763,E2 1729.763} C_VEL
LIN {X 0,Y 587.751,Z 675.537,A -85,B 0,C 180,E1 1732.732,E2 1732.732} C_VEL
LIN {X 0,Y 588.46,Z 641.437,A -85,B 0,C 180,E1 1735.335,E2 1735.335} C_VEL
LIN {X 0,Y 589.152,Z 606.147,A -85,B 0,C 180,E1 1737.337,E2 1737.337} C_VEL
LIN {X 0,Y 589.715,Z 570.367,A -85,B 0,C 180,E1 1738.778,E2 1738.778} C_VEL
LIN {X 0,Y 590.236,Z 532.26,A -85,B 0,C 180,E1 1739.728,E2 1739.728} C_VEL
LIN {X 0,Y 589.17,Z 484.125,A -85,B 0,C 180,E1 1740.478,E2 1740.478} C_VEL
LIN {X 0,Y 586.09,Z 476.03,A -85,B 0,C 180,E1 1740.789,E2 1740.789} C_VEL
LIN {X 0,Y 585.859,Z 476.03,A -85,B 0,C 180,E1 1746.767,E2 1746.767} C_VEL
LIN {X 0,Y 585.896,Z 476.03,A -85,B 0,C 180,E1 1752.214,E2 1752.214} C_VEL
LIN {X 0,Y 585.724,Z 476.03,A -85,B 0,C 180,E1 1757.777,E2 1757.777} C_VEL
LIN {X 0,Y 585.726,Z 476.03,A -85,B 0,C 180,E1 1763.26,E2 1763.26} C_VEL
LIN {X 0,Y 585.896,Z 476.03,A -85,B 0,C 180,E1 1768.518,E2 1768.518} C_VEL
LIN {X 0,Y 585.804,Z 476.03,A -85,B 0,C 180,E1 1773.939,E2 1773.939} C_VEL
LIN {X 0,Y 585.807,Z 476.03,A -85,B 0,C 180,E1 1778.79,E2 1778.79} C_VEL
LIN {X 0,Y 585.991,Z 476.03,A -85,B 0,C 180,E1 1783.491,E2 1783.491} C_VEL
LIN {X 0,Y 586.065,Z 476.03,A -85,B 0,C 180,E1 1788.075,E2 1788.075} C_VEL
LIN {X 0,Y 586.08,Z 476.03,A -85,B 0,C 180,E1 1792.581,E2 1792.581} C_VEL
LIN {X 0,Y 586.233,Z 476.03,A -85,B 0,C 180,E1 1797.042,E2 1797.042} C_VEL
LIN {X 0,Y 586.325,Z 476.03,A -85,B 0,C 180,E1 1801.482,E2 1801.482} C_VEL
LIN {X 0,Y 586.329,Z 476.03,A -85,B 0,C 180,E1 1805.931,E2 1805.931} C_VEL
LIN {X 0,Y 585.993,Z 476.03,A -85,B 0,C 180,E1 1811.931,E2 1811.931} C_VEL
LIN {X 0,Y 585.873,Z 476.03,A -85,B 0,C 180,E1 1817.018,E2 1817.018} C_VEL
LIN {X 0,Y 585.956,Z 476.03,A -85,B 0,C 180,E1 1821.528,E2 1821.528} C_VEL
LIN {X 0,Y 586.007,Z 476.03,A -85,B 0,C 180,E1 1826.056,E2 1826.056} C_VEL
LIN {X 0,Y 585.834,Z 476.03,A -85,B 0,C 180,E1 1831.472,E2 1831.472} C_VEL
LIN {X 0,Y 585.959,Z 476.03,A -85,B 0,C 180,E1 1836.771,E2 1836.771} C_VEL
LIN {X 0,Y 585.745,Z 476.03,A -85,B 0,C 180,E1 1842.227,E2 1842.227} C_VEL
LIN {X 0,Y 585.923,Z 476.03,A -85,B 0,C 180,E1 1847.788,E2 1847.788} C_VEL
LIN {X 0,Y 585.841,Z 476.03,A -85,B 0,C 180,E1 1853.528,E2 1853.528} C_VEL
LIN {X 0,Y 585.811,Z 476.03,A -85,B 0,C 180,E1 1858.874,E2 1858.874} C_VEL
LIN {X 0,Y 586.011,Z 476.03,A -85,B 0,C 180,E1 1864.728,E2 1864.728} C_VEL
LIN {X 0,Y 586.089,Z 476.03,A -85,B 0,C 180,E1 1870.376,E2 1870.376} C_VEL
LIN {X 0,Y 585.966,Z 476.03,A -85,B 0,C 180,E1 1876.553,E2 1876.553} C_VEL
LIN {X 0,Y 586.043,Z 476.03,A -85,B 0,C 180,E1 1877.266,E2 1877.266} C_VEL
LIN {X 0,Y 589.717,Z 487.611,A -85,B 0,C 180,E1 1877.785,E2 1877.785} C_VEL
LIN {X 0,Y 589.25,Z 527.566,A -85,B 0,C 180,E1 1879.217,E2 1879.217} C_VEL
LIN {X 0,Y 588.591,Z 565.187,A -85,B 0,C 180,E1 1881.215,E2 1881.215} C_VEL
LIN {X 0,Y 587.86,Z 600.684,A -85,B 0,C 180,E1 1883.805,E2 1883.805} C_VEL
LIN {X 0,Y 587.257,Z 632.186,A -85,B 0,C 180,E1 1886.86,E2 1886.86} C_VEL
LIN {X 0,Y 586.822,Z 658.33,A -85,B 0,C 180,E1 1890.185,E2 1890.185} C_VEL
LIN {X 0,Y 586.556,Z 679.191,A -85,B 0,C 180,E1 1893.7,E2 1893.7} C_VEL
LIN {X 0,Y 586.41,Z 695.062,A -85,B 0,C 180,E1 1897.418,E2 1897.418} C_VEL
LIN {X 0,Y 586.361,Z 705.39,A -85,B 0,C 180,E1 1901.124,E2 1901.124} C_VEL
LIN {X 0,Y 586.282,Z 710.74,A -85,B 0,C 180,E1 1904.967,E2 1904.967} C_VEL
LIN {X 0,Y 586.32,Z 711.258,A -85,B 0,C 180,E1 1908.053,E2 1908.053} C_VEL
LIN {X 0,Y 586.273,Z 707.599,A -85,B 0,C 180,E1 1911.61,E2 1911.61} C_VEL
LIN {X 0,Y 586.36,Z 698.816,A -85,B 0,C 180,E1 1915.344,E2 1915.344} C_VEL
LIN {X 0,Y 586.493,Z 685.155,A -85,B 0,C 180,E1 1918.967,E2 1918.967} C_VEL
LIN {X 0,Y 586.693,Z 665.339,A -85,B 0,C 180,E1 1922.656,E2 1922.656} C_VEL
LIN {X 0,Y 587.032,Z 642.056,A -85,B 0,C 180,E1 1925.901,E2 1925.901} C_VEL
LIN {X 0,Y 587.584,Z 613.645,A -85,B 0,C 180,E1 1928.947,E2 1928.947} C_VEL
LIN {X 0,Y 588.275,Z 581.59,A -85,B 0,C 180,E1 1931.59,E2 1931.59} C_VEL
LIN {X 0,Y 588.946,Z 546.024,A -85,B 0,C 180,E1 1933.797,E2 1933.797} C_VEL
LIN {X 0,Y 589.584,Z 508.89,A -85,B 0,C 180,E1 1935.439,E2 1935.439} C_VEL
LIN {X 0,Y 588.983,Z 484.596,A -85,B 0,C 180,E1 1936.245,E2 1936.245} C_VEL
LIN {X 0,Y 585.871,Z 476.03,A -85,B 0,C 180,E1 1936.705,E2 1936.705} C_VEL
LIN {X 0,Y 585.764,Z 476.03,A -85,B 0,C 180,E1 1941.658,E2 1941.658} C_VEL
LIN {X 0,Y 586.002,Z 476.03,A -85,B 0,C 180,E1 1947.139,E2 1947.139} C_VEL
LIN {X 0,Y 585.928,Z 476.03,A -85,B 0,C 180,E1 1952.28,E2 1952.28} C_VEL
LIN {X 0,Y 585.858,Z 476.03,A -85,B 0,C 180,E1 1958.498,E2 1958.498} C_VEL
LIN {X 0,Y 586.04,Z 476.372,A -85,B 0,C 180,E1 1962.291,E2 1962.291} C_VEL
LIN {X 0,Y 587.679,Z 498.919,A -85,B 0,C 180,E1 1962.811,E2 1962.811} C_VEL
LIN {X 0,Y 587.432,Z 528.596,A -85,B 0,C 180,E1 1963.913,E2 1963.913} C_VEL
LIN {X 0,Y 587.082,Z 556.849,A -85,B 0,C 180,E1 1965.587,E2 1965.587} C_VEL
LIN {X 0,Y 586.847,Z 581.316,A -85,B 0,C 180,E1 1967.709,E2 1967.709} C_VEL
LIN {X 0,Y 586.645,Z 601.14,A -85,B 0,C 180,E1 1970.153,E2 1970.153} C_VEL
LIN {X 0,Y 586.473,Z 616.8,A -85,B 0,C 180,E1 1972.989,E2 1972.989} C_VEL
LIN {X 0,Y 586.441,Z 625.739,A -85,B 0,C 180,E1 1975.556,E2 1975.556} C_VEL
LIN {X 0,Y 586.403,Z 630.89,A -85,B 0,C 180,E1 1978.518,E2 1978.518} C_VEL
LIN {X 0,Y 586.403,Z 630.815,A -85,B 0,C 180,E1 1981.477,E2 1981.477} C_VEL
LIN {X 0,Y 586.469,Z 627.476,A -85,B 0,C 180,E1 1983.635,E2 1983.635} C_VEL
LIN {X 0,Y 584.023,Z 624.485,A -85,B 0,C 180,E1 1984.864,E2 1984.864} C_VEL
LIN {X 0,Y 578.697,Z 618.301,A -85,B 0,C 180,E1 1986.652,E2 1986.652} C_VEL
LIN {X 0,Y 578.61,Z 617.463,A -85,B 0,C 180,E1 1986.854,E2 1986.854} C_VEL
LIN {X 0,Y 578.795,Z 601.818,A -85,B 0,C 180,E1 1989.787,E2 1989.787} C_VEL
LIN {X 0,Y 579.047,Z 582.308,A -85,B 0,C 180,E1 1992.263,E2 1992.263} C_VEL
LIN {X 0,Y 579.387,Z 558.195,A -85,B 0,C 180,E1 1994.419,E2 1994.419} C_VEL
LIN {X 0,Y 579.809,Z 530.769,A -85,B 0,C 180,E1 1996.105,E2 1996.105} C_VEL
LIN {X 0,Y 580.175,Z 499.466,A -85,B 0,C 180,E1 1997.313,E2 1997.313} C_VEL
LIN {X 0,Y 579.275,Z 480.495,A -85,B 0,C 180,E1 1997.766,E2 1997.766} C_VEL
LIN {X 0,Y 578.32,Z 476.03,A -85,B 0,C 180,E1 1997.915,E2 1997.915} C_VEL
LIN {X 0,Y 577.978,Z 476.03,A -85,B 0,C 180,E1 2003.524,E2 2003.524} C_VEL
LIN {X 0,Y 577.884,Z 476.03,A -85,B 0,C 180,E1 2008.135,E2 2008.135} C_VEL
LIN {X 0,Y 577.807,Z 476.03,A -85,B 0,C 180,E1 2013.382,E2 2013.382} C_VEL
LIN {X 0,Y 577.923,Z 476.03,A -85,B 0,C 180,E1 2018.954,E2 2018.954} C_VEL
LIN {X 0,Y 577.955,Z 476.03,A -85,B 0,C 180,E1 2024.981,E2 2024.981} C_VEL
LIN {X 0,Y 577.885,Z 476.03,A -85,B 0,C 180,E1 2031.036,E2 2031.036} C_VEL
LIN {X 0,Y 578.157,Z 476.03,A -85,B 0,C 180,E1 2036.923,E2 2036.923} C_VEL
LIN {X 0,Y 578.194,Z 476.03,A -85,B 0,C 180,E1 2038.741,E2 2038.741} C_VEL
LIN {X 0,Y 582.747,Z 487.563,A -85,B 0,C 180,E1 2039.198,E2 2039.198} C_VEL
LIN {X 0,Y 582.994,Z 549.201,A -85,B 0,C 180,E1 2040.231,E2 2040.231} C_VEL
LIN {X 0,Y 582.453,Z 588.458,A -85,B 0,C 180,E1 2041.508,E2 2041.508} C_VEL
LIN {X 0,Y 581.559,Z 625.717,A -85,B 0,C 180,E1 2043.338,E2 2043.338} C_VEL
LIN {X 0,Y 580.648,Z 661.541,A -85,B 0,C 180,E1 2045.784,E2 2045.784} C_VEL
LIN {X 0,Y 579.841,Z 692.245,A -85,B 0,C 180,E1 2048.557,E2 2048.557} C_VEL
LIN {X 0,Y 579.211,Z 719.24,A -85,B 0,C 180,E1 2051.718,E2 2051.718} C_VEL
LIN {X 0,Y 578.818,Z 741.893,A -85,B 0,C 180,E1 2055.191,E2 2055.191} C_VEL
LIN {X 0,Y 578.527,Z 758.792,A -85,B 0,C 180,E1 2058.669,E2 2058.669} C_VEL
LIN {X 0,Y 578.442,Z 771.625,A -85,B 0,C 180,E1 2062.479,E2 2062.479} C_VEL
LIN {X 0,Y 578.351,Z 777.942,A -85,B 0,C 180,E1 2065.495,E2 2065.495} C_VEL
LIN {X 0,Y 578.369,Z 781.09,A -85,B 0,C 180,E1 2068.5,E2 2068.5} C_VEL
LIN {X 0,Y 578.531,Z 781.091,A -85,B 0,C 180,E1 2071.499,E2 2071.499} C_VEL
LIN {X 0,Y 578.366,Z 776.81,A -85,B 0,C 180,E1 2075.209,E2 2075.209} C_VEL
LIN {X 0,Y 578.451,Z 767.22,A -85,B 0,C 180,E1 2079.036,E2 2079.036} C_VEL
LIN {X 0,Y 578.605,Z 752.089,A -85,B 0,C 180,E1 2082.852,E2 2082.852} C_VEL
LIN {X 0,Y 578.934,Z 731.569,A -85,B 0,C 180,E1 2086.524,E2 2086.524} C_VEL
LIN {X 0,Y 579.525,Z 705.356,A -85,B 0,C 180,E1 2090.016,E2 2090.016} C_VEL
LIN {X 0,Y 580.244,Z 675.542,A -85,B 0,C 180,E1 2093.042,E2 2093.042} C_VEL
LIN {X 0,Y 581.123,Z 642.203,A -85,B 0,C 180,E1 2095.626,E2 2095.626} C_VEL
LIN {X 0,Y 582.004,Z 606.573,A -85,B 0,C 180,E1 2097.681,E2 2097.681} C_VEL
LIN {X 0,Y 582.721,Z 570.076,A -85,B 0,C 180,E1 2099.166,E2 2099.166} C_VEL
LIN {X 0,Y 583.377,Z 532.215,A -85,B 0,C 180,E1 2100.115,E2 2100.115} C_VEL
LIN {X 0,Y 582.402,Z 486.591,A -85,B 0,C 180,E1 2100.836,E2 2100.836} C_VEL
LIN {X 0,Y 578.038,Z 476.03,A -85,B 0,C 180,E1 2101.303,E2 2101.303} C_VEL
LIN {X 0,Y 577.94,Z 476.03,A -85,B 0,C 180,E1 2107.054,E2 2107.054} C_VEL
LIN {X 0,Y 577.955,Z 476.03,A -85,B 0,C 180,E1 2112.933,E2 2112.933} C_VEL
LIN {X 0,Y 577.829,Z 476.03,A -85,B 0,C 180,E1 2119.08,E2 2119.08} C_VEL
LIN {X 0,Y 577.871,Z 476.03,A -85,B 0,C 180,E1 2124.806,E2 2124.806} C_VEL
LIN {X 0,Y 577.942,Z 476.03,A -85,B 0,C 180,E1 2130.153,E2 2130.153} C_VEL
LIN {X 0,Y 577.928,Z 476.03,A -85,B 0,C 180,E1 2135.221,E2 2135.221} C_VEL
LIN {X 0,Y 578.053,Z 476.03,A -85,B 0,C 180,E1 2140.554,E2 2140.554} C_VEL
LIN {X 0,Y 578.22,Z 476.03,A -85,B 0,C 180,E1 2146.372,E2 2146.372} C_VEL
LIN {X 0,Y 578.182,Z 476.03,A -85,B 0,C 180,E1 2152.479,E2 2152.479} C_VEL
LIN {X 0,Y 578.325,Z 476.03,A -85,B 0,C 180,E1 2157.001,E2 2157.001} C_VEL
LIN {X 0,Y 578.415,Z 476.03,A -85,B 0,C 180,E1 2161.502,E2 2161.502} C_VEL
LIN {X 0,Y 578.415,Z 476.03,A -85,B 0,C 180,E1 2166.012,E2 2166.012} C_VEL
LIN {X 0,Y 578.064,Z 476.03,A -85,B 0,C 180,E1 2172.097,E2 2172.097} C_VEL
LIN {X 0,Y 578.027,Z 476.03,A -85,B 0,C 180,E1 2176.748,E2 2176.748} C_VEL
LIN {X 0,Y 578.067,Z 476.03,A -85,B 0,C 180,E1 2181.513,E2 2181.513} C_VEL
LIN {X 0,Y 577.948,Z 476.03,A -85,B 0,C 180,E1 2187.035,E2 2187.035} C_VEL
LIN {X 0,Y 577.927,Z 476.03,A -85,B 0,C 180,E1 2191.6,E2 2191.6} C_VEL
LIN {X 0,Y 578.047,Z 476.03,A -85,B 0,C 180,E1 2197.046,E2 2197.046} C_VEL
LIN {X 0,Y 577.858,Z 476.03,A -85,B 0,C 180,E1 2202.941,E2 2202.941} C_VEL
LIN {X 0,Y 577.995,Z 476.03,A -85,B 0,C 180,E1 2207.178,E2 2207.178} C_VEL
LIN {X 0,Y 577.935,Z 476.03,A -85,B 0,C 180,E1 2212.946,E2 2212.946} C_VEL
LIN {X 0,Y 577.874,Z 476.03,A -85,B 0,C 180,E1 2218.397,E2 2218.397} C_VEL
LIN {X 0,Y 577.995,Z 476.03,A -85,B 0,C 180,E1 2223.556,E2 2223.556} C_VEL
LIN {X 0,Y 578.05,Z 476.03,A -85,B 0,C 180,E1 2228.487,E2 2228.487} C_VEL
LIN {X 0,Y 578.084,Z 476.03,A -85,B 0,C 180,E1 2233.255,E2 2233.255} C_VEL
LIN {X 0,Y 578.094,Z 476.03,A -85,B 0,C 180,E1 2236.828,E2 2236.828} C_VEL
LIN {X 0,Y 582.769,Z 490.724,A -85,B 0,C 180,E1 2237.49,E2 2237.49} C_VEL
LIN {X 0,Y 582.15,Z 530.736,A -85,B 0,C 180,E1 2238.992,E2 2238.992} C_VEL
LIN {X 0,Y 581.216,Z 568.96,A -85,B 0,C 180,E1 2241.112,E2 2241.112} C_VEL
LIN {X 0,Y 580.332,Z 602.333,A -85,B 0,C 180,E1 2243.634,E2 2243.634} C_VEL
LIN {X 0,Y 579.618,Z 632.61,A -85,B 0,C 180,E1 2246.631,E2 2246.631} C_VEL
LIN {X 0,Y 579.074,Z 658.647,A -85,B 0,C 180,E1 2250,E2 2250} C_VEL
LIN {X 0,Y 578.681,Z 680.39,A -85,B 0,C 180,E1 2253.751,E2 2253.751} C_VEL
LIN {X 0,Y 578.529,Z 695.885,A -85,B 0,C 180,E1 2257.52,E2 2257.52} C_VEL
LIN {X 0,Y 578.443,Z 705.877,A -85,B 0,C 180,E1 2261.278,E2 2261.278} C_VEL
LIN {X 0,Y 578.371,Z 710.902,A -85,B 0,C 180,E1 2265.177,E2 2265.177} C_VEL
LIN {X 0,Y 578.395,Z 711.183,A -85,B 0,C 180,E1 2268.309,E2 2268.309} C_VEL
LIN {X 0,Y 578.367,Z 707.208,A -85,B 0,C 180,E1 2271.921,E2 2271.921} C_VEL
LIN {X 0,Y 578.457,Z 698.039,A -85,B 0,C 180,E1 2275.716,E2 2275.716} C_VEL
LIN {X 0,Y 578.606,Z 683.785,A -85,B 0,C 180,E1 2279.435,E2 2279.435} C_VEL
LIN {X 0,Y 578.874,Z 665.117,A -85,B 0,C 180,E1 2282.91,E2 2282.91} C_VEL
LIN {X 0,Y 579.377,Z 640.393,A -85,B 0,C 180,E1 2286.367,E2 2286.367} C_VEL
LIN {X 0,Y 580.116,Z 611.348,A -85,B 0,C 180,E1 2289.468,E2 2289.468} C_VEL
LIN {X 0,Y 581.033,Z 577.38,A -85,B 0,C 180,E1 2292.227,E2 2292.227} C_VEL
LIN {X 0,Y 581.892,Z 541.732,A -85,B 0,C 180,E1 2294.382,E2 2294.382} C_VEL
LIN {X 0,Y 582.736,Z 503.409,A -85,B 0,C 180,E1 2296.011,E2 2296.011} C_VEL
LIN {X 0,Y 581.974,Z 487.316,A -85,B 0,C 180,E1 2296.559,E2 2296.559} C_VEL
LIN {X 0,Y 577.87,Z 476.03,A -85,B 0,C 180,E1 2297.128,E2 2297.128} C_VEL
LIN {X 0,Y 577.817,Z 476.03,A -85,B 0,C 180,E1 2302.937,E2 2302.937} C_VEL
LIN {X 0,Y 578.003,Z 476.03,A -85,B 0,C 180,E1 2308.405,E2 2308.405} C_VEL
LIN {X 0,Y 577.842,Z 476.03,A -85,B 0,C 180,E1 2313.547,E2 2313.547} C_VEL
LIN {X 0,Y 577.972,Z 476.03,A -85,B 0,C 180,E1 2318.483,E2 2318.483} C_VEL
LIN {X 0,Y 578.212,Z 476.03,A -85,B 0,C 180,E1 2322.023,E2 2322.023} C_VEL
LIN {X 0,Y 580.136,Z 498.886,A -85,B 0,C 180,E1 2322.58,E2 2322.58} C_VEL
LIN {X 0,Y 579.806,Z 528.583,A -85,B 0,C 180,E1 2323.695,E2 2323.695} C_VEL
LIN {X 0,Y 579.386,Z 556.673,A -85,B 0,C 180,E1 2325.379,E2 2325.379} C_VEL
LIN {X 0,Y 579.048,Z 581.306,A -85,B 0,C 180,E1 2327.541,E2 2327.541} C_VEL
LIN {X 0,Y 578.797,Z 601.133,A -85,B 0,C 180,E1 2330.018,E2 2330.018} C_VEL
LIN {X 0,Y 578.61,Z 616.65,A -85,B 0,C 180,E1 2332.858,E2 2332.858} C_VEL
LIN {X 0,Y 578.549,Z 625.74,A -85,B 0,C 180,E1 2335.495,E2 2335.495} C_VEL
LIN {X 0,Y 578.501,Z 630.891,A -85,B 0,C 180,E1 2338.498,E2 2338.498} C_VEL
LIN {X 0,Y 578.501,Z 630.813,A -85,B 0,C 180,E1 2341.497,E2 2341.497} C_VEL
LIN {X 0,Y 578.528,Z 625.525,A -85,B 0,C 180,E1 2344.501,E2 2344.501} C_VEL
LIN {X 0,Y 578.61,Z 617.463,A -85,B 0,C 180,E1 2346.854,E2 2346.854} C_VEL
LIN {X 0,Y 574.781,Z 610.401,A -85,B 0,C 180,E1 2348.402,E2 2348.402} C_VEL
LIN {X 0,Y 570.943,Z 601.974,A -85,B 0,C 180,E1 2349.899,E2 2349.899} C_VEL
LIN {X 0,Y 571.259,Z 582.31,A -85,B 0,C 180,E1 2352.433,E2 2352.433} C_VEL
LIN {X 0,Y 571.698,Z 557.076,A -85,B 0,C 180,E1 2354.7,E2 2354.7} C_VEL
LIN {X 0,Y 572.232,Z 528.81,A -85,B 0,C 180,E1 2356.423,E2 2356.423} C_VEL
LIN {X 0,Y 572.688,Z 497.439,A -85,B 0,C 180,E1 2357.606,E2 2357.606} C_VEL
LIN {X 0,Y 571.992,Z 482.773,A -85,B 0,C 180,E1 2357.959,E2 2357.959} C_VEL
LIN {X 0,Y 570.365,Z 476.03,A -85,B 0,C 180,E1 2358.144,E2 2358.144} C_VEL
LIN {X 0,Y 570.097,Z 476.03,A -85,B 0,C 180,E1 2363.473,E2 2363.473} C_VEL
LIN {X 0,Y 569.95,Z 476.03,A -85,B 0,C 180,E1 2368.756,E2 2368.756} C_VEL
LIN {X 0,Y 569.868,Z 476.03,A -85,B 0,C 180,E1 2374.547,E2 2374.547} C_VEL
LIN {X 0,Y 569.98,Z 476.03,A -85,B 0,C 180,E1 2379.613,E2 2379.613} C_VEL
LIN {X 0,Y 569.984,Z 476.03,A -85,B 0,C 180,E1 2384.173,E2 2384.173} C_VEL
LIN {X 0,Y 569.941,Z 476.03,A -85,B 0,C 180,E1 2390.387,E2 2390.387} C_VEL
LIN {X 0,Y 570.096,Z 476.03,A -85,B 0,C 180,E1 2396.1,E2 2396.1} C_VEL
LIN {X 0,Y 570.239,Z 476.03,A -85,B 0,C 180,E1 2398.263,E2 2398.263} C_VEL
LIN {X 0,Y 576.048,Z 490.453,A -85,B 0,C 180,E1 2398.841,E2 2398.841} C_VEL
LIN {X 0,Y 576.117,Z 548.639,A -85,B 0,C 180,E1 2399.826,E2 2399.826} C_VEL
LIN {X 0,Y 575.426,Z 588.548,A -85,B 0,C 180,E1 2401.132,E2 2401.132} C_VEL
LIN {X 0,Y 574.397,Z 625.245,A -85,B 0,C 180,E1 2402.95,E2 2402.95} C_VEL
LIN {X 0,Y 573.291,Z 660.449,A -85,B 0,C 180,E1 2405.363,E2 2405.363} C_VEL
LIN {X 0,Y 572.246,Z 692.249,A -85,B 0,C 180,E1 2408.258,E2 2408.258} C_VEL
LIN {X 0,Y 571.491,Z 720.356,A -85,B 0,C 180,E1 2411.613,E2 2411.613} C_VEL
LIN {X 0,Y 570.999,Z 743.127,A -85,B 0,C 180,E1 2415.205,E2 2415.205} C_VEL
LIN {X 0,Y 570.71,Z 760.6,A -85,B 0,C 180,E1 2418.965,E2 2418.965} C_VEL
LIN {X 0,Y 570.552,Z 771.628,A -85,B 0,C 180,E1 2422.375,E2 2422.375} C_VEL
LIN {X 0,Y 570.48,Z 777.944,A -85,B 0,C 180,E1 2425.433,E2 2425.433} C_VEL
LIN {X 0,Y 570.48,Z 781.092,A -85,B 0,C 180,E1 2428.479,E2 2428.479} C_VEL
LIN {X 0,Y 570.631,Z 781.093,A -85,B 0,C 180,E1 2431.52,E2 2431.52} C_VEL
LIN {X 0,Y 570.468,Z 777.031,A -85,B 0,C 180,E1 2435.148,E2 2435.148} C_VEL
LIN {X 0,Y 570.567,Z 767.223,A -85,B 0,C 180,E1 2439.161,E2 2439.161} C_VEL
LIN {X 0,Y 570.749,Z 752.093,A -85,B 0,C 180,E1 2443.032,E2 2443.032} C_VEL
LIN {X 0,Y 571.172,Z 731.57,A -85,B 0,C 180,E1 2446.755,E2 2446.755} C_VEL
LIN {X 0,Y 571.878,Z 705.025,A -85,B 0,C 180,E1 2450.334,E2 2450.334} C_VEL
LIN {X 0,Y 572.805,Z 674.266,A -85,B 0,C 180,E1 2453.475,E2 2453.475} C_VEL
LIN {X 0,Y 573.889,Z 641.047,A -85,B 0,C 180,E1 2456.053,E2 2456.053} C_VEL
LIN {X 0,Y 574.927,Z 604.744,A -85,B 0,C 180,E1 2458.144,E2 2458.144} C_VEL
LIN {X 0,Y 575.791,Z 568.297,A -85,B 0,C 180,E1 2459.61,E2 2459.61} C_VEL
LIN {X 0,Y 576.566,Z 530.066,A -85,B 0,C 180,E1 2460.544,E2 2460.544} C_VEL
LIN {X 0,Y 575.594,Z 489.044,A -85,B 0,C 180,E1 2461.207,E2 2461.207} C_VEL
LIN {X 0,Y 570.044,Z 476.03,A -85,B 0,C 180,E1 2461.803,E2 2461.803} C_VEL
LIN {X 0,Y 570.024,Z 476.03,A -85,B 0,C 180,E1 2467.657,E2 2467.657} C_VEL
LIN {X 0,Y 569.963,Z 476.03,A -85,B 0,C 180,E1 2473.685,E2 2473.685} C_VEL
LIN {X 0,Y 569.856,Z 476.03,A -85,B 0,C 180,E1 2478.382,E2 2478.382} C_VEL
LIN {X 0,Y 569.93,Z 476.03,A -85,B 0,C 180,E1 2484.241,E2 2484.241} C_VEL
LIN {X 0,Y 570.053,Z 476.03,A -85,B 0,C 180,E1 2489.697,E2 2489.697} C_VEL
LIN {X 0,Y 569.972,Z 476.03,A -85,B 0,C 180,E1 2494.852,E2 2494.852} C_VEL
LIN {X 0,Y 570.049,Z 476.03,A -85,B 0,C 180,E1 2499.804,E2 2499.804} C_VEL
LIN {X 0,Y 570.111,Z 476.03,A -85,B 0,C 180,E1 2504.602,E2 2504.602} C_VEL
LIN {X 0,Y 570.119,Z 476.03,A -85,B 0,C 180,E1 2509.308,E2 2509.308} C_VEL
LIN {X 0,Y 570.185,Z 476.03,A -85,B 0,C 180,E1 2513.905,E2 2513.905} C_VEL
LIN {X 0,Y 570.234,Z 476.03,A -85,B 0,C 180,E1 2518.481,E2 2518.481} C_VEL
LIN {X 0,Y 570.22,Z 476.03,A -85,B 0,C 180,E1 2523.046,E2 2523.046} C_VEL
LIN {X 0,Y 570.164,Z 476.03,A -85,B 0,C 180,E1 2527.632,E2 2527.632} C_VEL
LIN {X 0,Y 570.152,Z 476.03,A -85,B 0,C 180,E1 2532.267,E2 2532.267} C_VEL
LIN {X 0,Y 570.098,Z 476.03,A -85,B 0,C 180,E1 2537.037,E2 2537.037} C_VEL
LIN {X 0,Y 570.136,Z 476.03,A -85,B 0,C 180,E1 2541.827,E2 2541.827} C_VEL
LIN {X 0,Y 570.078,Z 476.03,A -85,B 0,C 180,E1 2546.842,E2 2546.842} C_VEL
LIN {X 0,Y 569.965,Z 476.03,A -85,B 0,C 180,E1 2552.094,E2 2552.094} C_VEL
LIN {X 0,Y 570.141,Z 476.03,A -85,B 0,C 180,E1 2557.648,E2 2557.648} C_VEL
LIN {X 0,Y 569.936,Z 476.03,A -85,B 0,C 180,E1 2564.169,E2 2564.169} C_VEL
LIN {X 0,Y 569.992,Z 476.03,A -85,B 0,C 180,E1 2568.387,E2 2568.387} C_VEL
LIN {X 0,Y 569.964,Z 476.03,A -85,B 0,C 180,E1 2574.237,E2 2574.237} C_VEL
LIN {X 0,Y 569.999,Z 476.03,A -85,B 0,C 180,E1 2579.688,E2 2579.688} C_VEL
LIN {X 0,Y 570.13,Z 476.03,A -85,B 0,C 180,E1 2584.855,E2 2584.855} C_VEL
LIN {X 0,Y 570.202,Z 476.03,A -85,B 0,C 180,E1 2589.806,E2 2589.806} C_VEL
LIN {X 0,Y 570.101,Z 476.03,A -85,B 0,C 180,E1 2594.598,E2 2594.598} C_VEL
LIN {X 0,Y 570.184,Z 476.738,A -85,B 0,C 180,E1 2596.384,E2 2596.384} C_VEL
LIN {X 0,Y 575.824,Z 492.82,A -85,B 0,C 180,E1 2597.166,E2 2597.166} C_VEL
LIN {X 0,Y 575.032,Z 532.551,A -85,B 0,C 180,E1 2598.707,E2 2598.707} C_VEL
LIN {X 0,Y 573.957,Z 569.505,A -85,B 0,C 180,E1 2600.797,E2 2600.797} C_VEL
LIN {X 0,Y 572.874,Z 602.128,A -85,B 0,C 180,E1 2603.294,E2 2603.294} C_VEL
LIN {X 0,Y 571.97,Z 633.039,A -85,B 0,C 180,E1 2606.396,E2 2606.396} C_VEL
LIN {X 0,Y 571.29,Z 658.97,A -85,B 0,C 180,E1 2609.81,E2 2609.81} C_VEL
LIN {X 0,Y 570.914,Z 679.656,A -85,B 0,C 180,E1 2613.421,E2 2613.421} C_VEL
LIN {X 0,Y 570.672,Z 695.37,A -85,B 0,C 180,E1 2617.24,E2 2617.24} C_VEL
LIN {X 0,Y 570.599,Z 705.376,A -85,B 0,C 180,E1 2620.953,E2 2620.953} C_VEL
LIN {X 0,Y 570.455,Z 709.806,A -85,B 0,C 180,E1 2623.821,E2 2623.821} C_VEL
LIN {X 0,Y 570.405,Z 711.466,A -85,B 0,C 180,E1 2627.143,E2 2627.143} C_VEL
LIN {X 0,Y 570.484,Z 708.792,A -85,B 0,C 180,E1 2630.959,E2 2630.959} C_VEL
LIN {X 0,Y 570.59,Z 700.168,A -85,B 0,C 180,E1 2635.124,E2 2635.124} C_VEL
LIN {X 0,Y 570.776,Z 686.887,A -85,B 0,C 180,E1 2638.91,E2 2638.91} C_VEL
LIN {X 0,Y 571.067,Z 667.04,A -85,B 0,C 180,E1 2642.819,E2 2642.819} C_VEL
LIN {X 0,Y 571.644,Z 643.552,A -85,B 0,C 180,E1 2646.245,E2 2646.245} C_VEL
LIN {X 0,Y 572.53,Z 613.877,A -85,B 0,C 180,E1 2649.535,E2 2649.535} C_VEL
LIN {X 0,Y 573.556,Z 582.367,A -85,B 0,C 180,E1 2652.208,E2 2652.208} C_VEL
LIN {X 0,Y 574.62,Z 546.709,A -85,B 0,C 180,E1 2654.484,E2 2654.484} C_VEL
LIN {X 0,Y 575.624,Z 509.824,A -85,B 0,C 180,E1 2656.16,E2 2656.16} C_VEL
LIN {X 0,Y 575.12,Z 490.015,A -85,B 0,C 180,E1 2656.873,E2 2656.873} C_VEL
LIN {X 0,Y 569.924,Z 476.03,A -85,B 0,C 180,E1 2657.61,E2 2657.61} C_VEL
LIN {X 0,Y 569.923,Z 476.03,A -85,B 0,C 180,E1 2662.846,E2 2662.846} C_VEL
LIN {X 0,Y 570.096,Z 476.03,A -85,B 0,C 180,E1 2668.2,E2 2668.2} C_VEL
LIN {X 0,Y 569.977,Z 476.03,A -85,B 0,C 180,E1 2673.153,E2 2673.153} C_VEL
LIN {X 0,Y 570.06,Z 476.03,A -85,B 0,C 180,E1 2678.377,E2 2678.377} C_VEL
LIN {X 0,Y 570.225,Z 476.03,A -85,B 0,C 180,E1 2681.752,E2 2681.752} C_VEL
LIN {X 0,Y 572.619,Z 497.538,A -85,B 0,C 180,E1 2682.305,E2 2682.305} C_VEL
LIN {X 0,Y 572.203,Z 528.57,A -85,B 0,C 180,E1 2683.472,E2 2683.472} C_VEL
LIN {X 0,Y 571.71,Z 556.661,A -85,B 0,C 180,E1 2685.178,E2 2685.178} C_VEL
LIN {X 0,Y 571.251,Z 581.296,A -85,B 0,C 180,E1 2687.368,E2 2687.368} C_VEL
LIN {X 0,Y 570.94,Z 601.126,A -85,B 0,C 180,E1 2689.879,E2 2689.879} C_VEL
LIN {X 0,Y 570.722,Z 616.644,A -85,B 0,C 180,E1 2692.759,E2 2692.759} C_VEL
LIN {X 0,Y 570.681,Z 625.74,A -85,B 0,C 180,E1 2695.433,E2 2695.433} C_VEL
LIN {X 0,Y 570.608,Z 630.891,A -85,B 0,C 180,E1 2698.477,E2 2698.477} C_VEL
LIN {X 0,Y 570.608,Z 630.811,A -85,B 0,C 180,E1 2701.518,E2 2701.518} C_VEL
LIN {X 0,Y 570.656,Z 625.529,A -85,B 0,C 180,E1 2704.563,E2 2704.563} C_VEL
LIN {X 0,Y 570.72,Z 614.53,A -85,B 0,C 180,E1 2707.62,E2 2707.62} C_VEL
LIN {X 0,Y 570.943,Z 601.974,A -85,B 0,C 180,E1 2709.899,E2 2709.899} C_VEL
LIN {X 0,Y 567.188,Z 592.431,A -85,B 0,C 180,E1 2711.332,E2 2711.332} C_VEL
LIN {X 0,Y 563.442,Z 581.62,A -85,B 0,C 180,E1 2712.683,E2 2712.683} C_VEL
LIN {X 0,Y 564.01,Z 557.356,A -85,B 0,C 180,E1 2714.885,E2 2714.885} C_VEL
LIN {X 0,Y 564.625,Z 528.817,A -85,B 0,C 180,E1 2716.651,E2 2716.651} C_VEL
LIN {X 0,Y 565.148,Z 498.103,A -85,B 0,C 180,E1 2717.831,E2 2717.831} C_VEL
LIN {X 0,Y 564.095,Z 482.84,A -85,B 0,C 180,E1 2718.218,E2 2718.218} C_VEL
LIN {X 0,Y 562.466,Z 476.03,A -85,B 0,C 180,E1 2718.459,E2 2718.459} C_VEL
LIN {X 0,Y 562.193,Z 476.03,A -85,B 0,C 180,E1 2723.823,E2 2723.823} C_VEL
LIN {X 0,Y 562.029,Z 476.03,A -85,B 0,C 180,E1 2729.002,E2 2729.002} C_VEL
LIN {X 0,Y 561.971,Z 476.03,A -85,B 0,C 180,E1 2734.452,E2 2734.452} C_VEL
LIN {X 0,Y 562.036,Z 476.03,A -85,B 0,C 180,E1 2740.276,E2 2740.276} C_VEL
LIN {X 0,Y 562.023,Z 476.03,A -85,B 0,C 180,E1 2745.536,E2 2745.536} C_VEL
LIN {X 0,Y 561.953,Z 476.03,A -85,B 0,C 180,E1 2751.705,E2 2751.705} C_VEL
LIN {X 0,Y 562.279,Z 476.03,A -85,B 0,C 180,E1 2757.749,E2 2757.749} C_VEL
LIN {X 0,Y 569.337,Z 494.679,A -85,B 0,C 180,E1 2758.493,E2 2758.493} C_VEL
LIN {X 0,Y 569.24,Z 550.294,A -85,B 0,C 180,E1 2759.465,E2 2759.465} C_VEL
LIN {X 0,Y 568.425,Z 589.07,A -85,B 0,C 180,E1 2760.764,E2 2760.764} C_VEL
LIN {X 0,Y 567.21,Z 625.248,A -85,B 0,C 180,E1 2762.58,E2 2762.58} C_VEL
LIN {X 0,Y 565.899,Z 660.727,A -85,B 0,C 180,E1 2765.042,E2 2765.042} C_VEL
LIN {X 0,Y 564.691,Z 692.253,A -85,B 0,C 180,E1 2767.952,E2 2767.952} C_VEL
LIN {X 0,Y 563.822,Z 719.248,A -85,B 0,C 180,E1 2771.2,E2 2771.2} C_VEL
LIN {X 0,Y 563.196,Z 741.47,A -85,B 0,C 180,E1 2774.692,E2 2774.692} C_VEL
LIN {X 0,Y 562.774,Z 758.841,A -85,B 0,C 180,E1 2778.358,E2 2778.358} C_VEL
LIN {X 0,Y 562.681,Z 771.631,A -85,B 0,C 180,E1 2782.267,E2 2782.267} C_VEL
LIN {X 0,Y 562.578,Z 777.947,A -85,B 0,C 180,E1 2785.369,E2 2785.369} C_VEL
LIN {X 0,Y 562.577,Z 781.095,A -85,B 0,C 180,E1 2788.457,E2 2788.457} C_VEL
LIN {X 0,Y 562.728,Z 781.095,A -85,B 0,C 180,E1 2791.542,E2 2791.542} C_VEL
LIN {X 0,Y 562.564,Z 776.904,A -85,B 0,C 180,E1 2795.301,E2 2795.301} C_VEL
LIN {X 0,Y 562.706,Z 767.226,A -85,B 0,C 180,E1 2799.291,E2 2799.291} C_VEL
LIN {X 0,Y 562.921,Z 752.096,A -85,B 0,C 180,E1 2803.216,E2 2803.216} C_VEL
LIN {X 0,Y 563.414,Z 731.57,A -85,B 0,C 180,E1 2806.993,E2 2806.993} C_VEL
LIN {X 0,Y 564.276,Z 705.029,A -85,B 0,C 180,E1 2810.621,E2 2810.621} C_VEL
LIN {X 0,Y 565.358,Z 674.428,A -85,B 0,C 180,E1 2813.789,E2 2813.789} C_VEL
LIN {X 0,Y 566.632,Z 641.053,A -85,B 0,C 180,E1 2816.413,E2 2816.413} C_VEL
LIN {X 0,Y 567.868,Z 604.725,A -85,B 0,C 180,E1 2818.527,E2 2818.527} C_VEL
LIN {X 0,Y 568.915,Z 566.341,A -85,B 0,C 180,E1 2820.071,E2 2820.071} C_VEL
LIN {X 0,Y 569.756,Z 526.427,A -85,B 0,C 180,E1 2821.012,E2 2821.012} C_VEL
LIN {X 0,Y 568.741,Z 491.421,A -85,B 0,C 180,E1 2821.591,E2 2821.591} C_VEL
LIN {X 0,Y 562.064,Z 476.03,A -85,B 0,C 180,E1 2822.265,E2 2822.265} C_VEL
LIN {X 0,Y 562.033,Z 476.03,A -85,B 0,C 180,E1 2828.288,E2 2828.288} C_VEL
LIN {X 0,Y 562.045,Z 476.03,A -85,B 0,C 180,E1 2834.461,E2 2834.461} C_VEL
LIN {X 0,Y 561.924,Z 476.03,A -85,B 0,C 180,E1 2839.715,E2 2839.715} C_VEL
LIN {X 0,Y 562.081,Z 476.03,A -85,B 0,C 180,E1 2845.555,E2 2845.555} C_VEL
LIN {X 0,Y 562.105,Z 476.03,A -85,B 0,C 180,E1 2851.002,E2 2851.002} C_VEL
LIN {X 0,Y 562.136,Z 476.03,A -85,B 0,C 180,E1 2856.318,E2 2856.318} C_VEL
LIN {X 0,Y 562.247,Z 476.03,A -85,B 0,C 180,E1 2861.15,E2 2861.15} C_VEL
LIN {X 0,Y 562.334,Z 476.03,A -85,B 0,C 180,E1 2867.564,E2 2867.564} C_VEL
LIN {X 0,Y 562.365,Z 476.03,A -85,B 0,C 180,E1 2872.266,E2 2872.266} C_VEL
LIN {X 0,Y 562.508,Z 476.03,A -85,B 0,C 180,E1 2876.917,E2 2876.917} C_VEL
LIN {X 0,Y 562.608,Z 476.03,A -85,B 0,C 180,E1 2881.544,E2 2881.544} C_VEL
LIN {X 0,Y 562.562,Z 476.03,A -85,B 0,C 180,E1 2886.182,E2 2886.182} C_VEL
LIN {X 0,Y 562.23,Z 476.03,A -85,B 0,C 180,E1 2892.443,E2 2892.443} C_VEL
LIN {X 0,Y 562.199,Z 476.03,A -85,B 0,C 180,E1 2897.234,E2 2897.234} C_VEL
LIN {X 0,Y 562.194,Z 476.03,A -85,B 0,C 180,E1 2902.152,E2 2902.152} C_VEL
LIN {X 0,Y 562.105,Z 476.03,A -85,B 0,C 180,E1 2907.265,E2 2907.265} C_VEL
LIN {X 0,Y 561.992,Z 476.03,A -85,B 0,C 180,E1 2912.605,E2 2912.605} C_VEL
LIN {X 0,Y 562.132,Z 476.03,A -85,B 0,C 180,E1 2918.28,E2 2918.28} C_VEL
LIN {X 0,Y 562.024,Z 476.03,A -85,B 0,C 180,E1 2924.462,E2 2924.462} C_VEL
LIN {X 0,Y 562.049,Z 476.03,A -85,B 0,C 180,E1 2929.719,E2 2929.719} C_VEL
LIN {X 0,Y 561.97,Z 476.03,A -85,B 0,C 180,E1 2935.542,E2 2935.542} C_VEL
LIN {X 0,Y 562.039,Z 476.03,A -85,B 0,C 180,E1 2940.993,E2 2940.993} C_VEL
LIN {X 0,Y 562.171,Z 476.03,A -85,B 0,C 180,E1 2946.307,E2 2946.307} C_VEL
LIN {X 0,Y 562.281,Z 476.03,A -85,B 0,C 180,E1 2951.148,E2 2951.148} C_VEL
LIN {X 0,Y 562.196,Z 476.109,A -85,B 0,C 180,E1 2955.887,E2 2955.887} C_VEL
LIN {X 0,Y 568.876,Z 495.743,A -85,B 0,C 180,E1 2956.86,E2 2956.86} C_VEL
LIN {X 0,Y 567.943,Z 533.473,A -85,B 0,C 180,E1 2958.369,E2 2958.369} C_VEL
LIN {X 0,Y 566.683,Z 570.203,A -85,B 0,C 180,E1 2960.484,E2 2960.484} C_VEL
LIN {X 0,Y 565.363,Z 604.472,A -85,B 0,C 180,E1 2963.175,E2 2963.175} C_VEL
LIN {X 0,Y 564.304,Z 635.124,A -85,B 0,C 180,E1 2966.347,E2 2966.347} C_VEL
LIN {X 0,Y 563.453,Z 661.792,A -85,B 0,C 180,E1 2970,E2 2970} C_VEL
LIN {X 0,Y 562.938,Z 682.611,A -85,B 0,C 180,E1 2973.856,E2 2973.856} C_VEL
LIN {X 0,Y 562.74,Z 697.403,A -85,B 0,C 180,E1 2977.732,E2 2977.732} C_VEL
LIN {X 0,Y 562.635,Z 706.876,A -85,B 0,C 180,E1 2981.645,E2 2981.645} C_VEL
LIN {X 0,Y 562.539,Z 711.2,A -85,B 0,C 180,E1 2985.614,E2 2985.614} C_VEL
LIN {X 0,Y 562.568,Z 710.326,A -85,B 0,C 180,E1 2989.614,E2 2989.614} C_VEL
LIN {X 0,Y 562.661,Z 703.776,A -85,B 0,C 180,E1 2993.807,E2 2993.807} C_VEL
LIN {X 0,Y 562.855,Z 692.172,A -85,B 0,C 180,E1 2997.733,E2 2997.733} C_VEL
LIN {X 0,Y 563.208,Z 674.044,A -85,B 0,C 180,E1 3001.789,E2 3001.789} C_VEL
LIN {X 0,Y 563.796,Z 651.241,A -85,B 0,C 180,E1 3005.477,E2 3005.477} C_VEL
LIN {X 0,Y 564.675,Z 623.592,A -85,B 0,C 180,E1 3008.86,E2 3008.86} C_VEL
LIN {X 0,Y 565.843,Z 591.871,A -85,B 0,C 180,E1 3011.817,E2 3011.817} C_VEL
LIN {X 0,Y 567.115,Z 556.941,A -85,B 0,C 180,E1 3014.277,E2 3014.277} C_VEL
LIN {X 0,Y 568.4,Z 517.974,A -85,B 0,C 180,E1 3016.238,E2 3016.238} C_VEL
LIN {X 0,Y 568.198,Z 492.521,A -85,B 0,C 180,E1 3017.195,E2 3017.195} C_VEL
LIN {X 0,Y 561.954,Z 476.03,A -85,B 0,C 180,E1 3018.092,E2 3018.092} C_VEL
LIN {X 0,Y 561.995,Z 476.03,A -85,B 0,C 180,E1 3023.926,E2 3023.926} C_VEL
LIN {X 0,Y 562.193,Z 476.03,A -85,B 0,C 180,E1 3029.524,E2 3029.524} C_VEL
LIN {X 0,Y 562.001,Z 476.03,A -85,B 0,C 180,E1 3034.464,E2 3034.464} C_VEL
LIN {X 0,Y 562.066,Z 476.03,A -85,B 0,C 180,E1 3039.5,E2 3039.5} C_VEL
LIN {X 0,Y 562.261,Z 476.03,A -85,B 0,C 180,E1 3041.509,E2 3041.509} C_VEL
LIN {X 0,Y 565.079,Z 498.715,A -85,B 0,C 180,E1 3042.098,E2 3042.098} C_VEL
LIN {X 0,Y 564.572,Z 528.557,A -85,B 0,C 180,E1 3043.242,E2 3043.242} C_VEL
LIN {X 0,Y 564.017,Z 557.484,A -85,B 0,C 180,E1 3045.034,E2 3045.034} C_VEL
LIN {X 0,Y 563.429,Z 583.09,A -85,B 0,C 180,E1 3047.387,E2 3047.387} C_VEL
LIN {X 0,Y 563.054,Z 603.589,A -85,B 0,C 180,E1 3050.127,E2 3050.127} C_VEL
LIN {X 0,Y 562.824,Z 618.216,A -85,B 0,C 180,E1 3053.045,E2 3053.045} C_VEL
LIN {X 0,Y 562.753,Z 627.529,A -85,B 0,C 180,E1 3056.141,E2 3056.141} C_VEL
LIN {X 0,Y 562.706,Z 630.89,A -85,B 0,C 180,E1 3058.456,E2 3058.456} C_VEL
LIN {X 0,Y 562.706,Z 630.809,A -85,B 0,C 180,E1 3061.539,E2 3061.539} C_VEL
LIN {X 0,Y 562.759,Z 625.533,A -85,B 0,C 180,E1 3064.627,E2 3064.627} C_VEL
LIN {X 0,Y 562.844,Z 614.535,A -85,B 0,C 180,E1 3067.727,E2 3067.727} C_VEL
LIN {X 0,Y 563.156,Z 597.913,A -85,B 0,C 180,E1 3070.649,E2 3070.649} C_VEL
LIN {X 0,Y 563.442,Z 581.62,A -85,B 0,C 180,E1 3072.683,E2 3072.683} C_VEL
LIN {X 0,Y 559.785,Z 569.83,A -85,B 0,C 180,E1 3073.959,E2 3073.959} C_VEL
LIN {X 0,Y 556.317,Z 556.958,A -85,B 0,C 180,E1 3075.126,E2 3075.126} C_VEL
LIN {X 0,Y 557.019,Z 528.824,A -85,B 0,C 180,E1 3076.885,E2 3076.885} C_VEL
LIN {X 0,Y 557.637,Z 498.162,A -85,B 0,C 180,E1 3078.079,E2 3078.079} C_VEL
LIN {X 0,Y 556.687,Z 484.773,A -85,B 0,C 180,E1 3078.43,E2 3078.43} C_VEL
LIN {X 0,Y 554.547,Z 476.03,A -85,B 0,C 180,E1 3078.651,E2 3078.651} C_VEL
LIN {X 0,Y 554.26,Z 476.03,A -85,B 0,C 180,E1 3084.186,E2 3084.186} C_VEL
LIN {X 0,Y 554.107,Z 476.03,A -85,B 0,C 180,E1 3089.458,E2 3089.458} C_VEL
LIN {X 0,Y 554.079,Z 476.03,A -85,B 0,C 180,E1 3095.014,E2 3095.014} C_VEL
LIN {X 0,Y 554.129,Z 476.03,A -85,B 0,C 180,E1 3100.972,E2 3100.972} C_VEL
LIN {X 0,Y 554.079,Z 476.03,A -85,B 0,C 180,E1 3106.908,E2 3106.908} C_VEL
LIN {X 0,Y 554.023,Z 476.03,A -85,B 0,C 180,E1 3113.04,E2 3113.04} C_VEL
LIN {X 0,Y 554.314,Z 476.03,A -85,B 0,C 180,E1 3117.237,E2 3117.237} C_VEL
LIN {X 0,Y 562.642,Z 496.959,A -85,B 0,C 180,E1 3118.108,E2 3118.108} C_VEL
LIN {X 0,Y 562.41,Z 550.767,A -85,B 0,C 180,E1 3119.067,E2 3119.067} C_VEL
LIN {X 0,Y 561.44,Z 589.303,A -85,B 0,C 180,E1 3120.375,E2 3120.375} C_VEL
LIN {X 0,Y 560.018,Z 626.402,A -85,B 0,C 180,E1 3122.269,E2 3122.269} C_VEL
LIN {X 0,Y 558.522,Z 661.154,A -85,B 0,C 180,E1 3124.725,E2 3124.725} C_VEL
LIN {X 0,Y 557.13,Z 692.257,A -85,B 0,C 180,E1 3127.636,E2 3127.636} C_VEL
LIN {X 0,Y 556.098,Z 719.252,A -85,B 0,C 180,E1 3130.929,E2 3130.929} C_VEL
LIN {X 0,Y 555.38,Z 741.284,A -85,B 0,C 180,E1 3134.437,E2 3134.437} C_VEL
LIN {X 0,Y 554.913,Z 758.845,A -85,B 0,C 180,E1 3138.191,E2 3138.191} C_VEL
LIN {X 0,Y 554.789,Z 771.634,A -85,B 0,C 180,E1 3142.157,E2 3142.157} C_VEL
LIN {X 0,Y 554.687,Z 777.95,A -85,B 0,C 180,E1 3145.302,E2 3145.302} C_VEL
LIN {X 0,Y 554.675,Z 781.097,A -85,B 0,C 180,E1 3148.436,E2 3148.436} C_VEL
LIN {X 0,Y 554.824,Z 781.097,A -85,B 0,C 180,E1 3151.564,E2 3151.564} C_VEL
LIN {X 0,Y 554.666,Z 776.903,A -85,B 0,C 180,E1 3155.377,E2 3155.377} C_VEL
LIN {X 0,Y 554.821,Z 767.229,A -85,B 0,C 180,E1 3159.424,E2 3159.424} C_VEL
LIN {X 0,Y 555.085,Z 752.099,A -85,B 0,C 180,E1 3163.406,E2 3163.406} C_VEL
LIN {X 0,Y 555.69,Z 731.568,A -85,B 0,C 180,E1 3167.236,E2 3167.236} C_VEL
LIN {X 0,Y 556.7,Z 705.032,A -85,B 0,C 180,E1 3170.914,E2 3170.914} C_VEL
LIN {X 0,Y 557.897,Z 675.558,A -85,B 0,C 180,E1 3174.022,E2 3174.022} C_VEL
LIN {X 0,Y 559.358,Z 641.851,A -85,B 0,C 180,E1 3176.727,E2 3176.727} C_VEL
LIN {X 0,Y 560.778,Z 606.331,A -85,B 0,C 180,E1 3178.838,E2 3178.838} C_VEL
LIN {X 0,Y 562,Z 568.034,A -85,B 0,C 180,E1 3180.422,E2 3180.422} C_VEL
LIN {X 0,Y 562.987,Z 528.277,A -85,B 0,C 180,E1 3181.395,E2 3181.395} C_VEL
LIN {X 0,Y 562.001,Z 493.888,A -85,B 0,C 180,E1 3181.978,E2 3181.978} C_VEL
LIN {X 0,Y 554.107,Z 476.03,A -85,B 0,C 180,E1 3182.799,E2 3182.799} C_VEL
LIN {X 0,Y 554.113,Z 476.03,A -85,B 0,C 180,E1 3188.937,E2 3188.937} C_VEL
LIN {X 0,Y 554.139,Z 476.03,A -85,B 0,C 180,E1 3194.739,E2 3194.739} C_VEL
LIN {X 0,Y 554.019,Z 476.03,A -85,B 0,C 180,E1 3201.061,E2 3201.061} C_VEL
LIN {X 0,Y 554.233,Z 476.03,A -85,B 0,C 180,E1 3206.886,E2 3206.886} C_VEL
LIN {X 0,Y 554.109,Z 476.03,A -85,B 0,C 180,E1 3212.325,E2 3212.325} C_VEL
LIN {X 0,Y 554.178,Z 476.03,A -85,B 0,C 180,E1 3218.27,E2 3218.27} C_VEL
LIN {X 0,Y 554.403,Z 476.03,A -85,B 0,C 180,E1 3222.915,E2 3222.915} C_VEL
LIN {X 0,Y 554.413,Z 476.03,A -85,B 0,C 180,E1 3227.384,E2 3227.384} C_VEL
LIN {X 0,Y 554.45,Z 476.03,A -85,B 0,C 180,E1 3232.155,E2 3232.155} C_VEL
LIN {X 0,Y 554.62,Z 476.03,A -85,B 0,C 180,E1 3236.873,E2 3236.873} C_VEL
LIN {X 0,Y 554.698,Z 476.03,A -85,B 0,C 180,E1 3241.566,E2 3241.566} C_VEL
LIN {X 0,Y 554.631,Z 476.03,A -85,B 0,C 180,E1 3246.271,E2 3246.271} C_VEL
LIN {X 0,Y 554.308,Z 476.03,A -85,B 0,C 180,E1 3252.624,E2 3252.624} C_VEL
LIN {X 0,Y 554.282,Z 476.03,A -85,B 0,C 180,E1 3257.488,E2 3257.488} C_VEL
LIN {X 0,Y 554.271,Z 476.03,A -85,B 0,C 180,E1 3262.486,E2 3262.486} C_VEL
LIN {X 0,Y 554.179,Z 476.03,A -85,B 0,C 180,E1 3267.676,E2 3267.676} C_VEL
LIN {X 0,Y 554.085,Z 476.03,A -85,B 0,C 180,E1 3273.129,E2 3273.129} C_VEL
LIN {X 0,Y 554.187,Z 476.03,A -85,B 0,C 180,E1 3278.931,E2 3278.931} C_VEL
LIN {X 0,Y 554.168,Z 476.03,A -85,B 0,C 180,E1 3285.265,E2 3285.265} C_VEL
LIN {X 0,Y 554.124,Z 476.03,A -85,B 0,C 180,E1 3291.063,E2 3291.063} C_VEL
LIN {X 0,Y 554.042,Z 476.03,A -85,B 0,C 180,E1 3296.868,E2 3296.868} C_VEL
LIN {X 0,Y 554.157,Z 476.03,A -85,B 0,C 180,E1 3302.323,E2 3302.323} C_VEL
LIN {X 0,Y 554.27,Z 476.03,A -85,B 0,C 180,E1 3308.243,E2 3308.243} C_VEL
LIN {X 0,Y 554.357,Z 476.03,A -85,B 0,C 180,E1 3312.926,E2 3312.926} C_VEL
LIN {X 0,Y 554.298,Z 476.213,A -85,B 0,C 180,E1 3315.396,E2 3315.396} C_VEL
LIN {X 0,Y 561.927,Z 498.256,A -85,B 0,C 180,E1 3316.535,E2 3316.535} C_VEL
LIN {X 0,Y 560.796,Z 536.342,A -85,B 0,C 180,E1 3318.12,E2 3318.12} C_VEL
LIN {X 0,Y 559.37,Z 572.304,A -85,B 0,C 180,E1 3320.26,E2 3320.26} C_VEL
LIN {X 0,Y 557.885,Z 605.357,A -85,B 0,C 180,E1 3322.919,E2 3322.919} C_VEL
LIN {X 0,Y 556.67,Z 635.531,A -85,B 0,C 180,E1 3326.101,E2 3326.101} C_VEL
LIN {X 0,Y 555.687,Z 662.087,A -85,B 0,C 180,E1 3329.805,E2 3329.805} C_VEL
LIN {X 0,Y 555.172,Z 681.927,A -85,B 0,C 180,E1 3333.518,E2 3333.518} C_VEL
LIN {X 0,Y 554.91,Z 696.958,A -85,B 0,C 180,E1 3337.447,E2 3337.447} C_VEL
LIN {X 0,Y 554.813,Z 705.841,A -85,B 0,C 180,E1 3341.013,E2 3341.013} C_VEL
LIN {X 0,Y 554.636,Z 710.296,A -85,B 0,C 180,E1 3344.223,E2 3344.223} C_VEL
LIN {X 0,Y 554.593,Z 711.396,A -85,B 0,C 180,E1 3347.477,E2 3347.477} C_VEL
LIN {X 0,Y 554.679,Z 709.153,A -85,B 0,C 180,E1 3350.785,E2 3350.785} C_VEL
LIN {X 0,Y 554.836,Z 701.224,A -85,B 0,C 180,E1 3354.961,E2 3354.961} C_VEL
LIN {X 0,Y 555.04,Z 687.095,A -85,B 0,C 180,E1 3359.2,E2 3359.2} C_VEL
LIN {X 0,Y 555.447,Z 668.425,A -85,B 0,C 180,E1 3363.038,E2 3363.038} C_VEL
LIN {X 0,Y 556.297,Z 643.681,A -85,B 0,C 180,E1 3366.784,E2 3366.784} C_VEL
LIN {X 0,Y 557.499,Z 615.134,A -85,B 0,C 180,E1 3370.052,E2 3370.052} C_VEL
LIN {X 0,Y 558.899,Z 583.158,A -85,B 0,C 180,E1 3372.858,E2 3372.858} C_VEL
LIN {X 0,Y 560.39,Z 547.253,A -85,B 0,C 180,E1 3375.214,E2 3375.214} C_VEL
LIN {X 0,Y 561.653,Z 512.189,A -85,B 0,C 180,E1 3376.865,E2 3376.865} C_VEL
LIN {X 0,Y 561.425,Z 495.564,A -85,B 0,C 180,E1 3377.495,E2 3377.495} C_VEL
LIN {X 0,Y 554.033,Z 476.03,A -85,B 0,C 180,E1 3378.641,E2 3378.641} C_VEL
LIN {X 0,Y 554.125,Z 476.03,A -85,B 0,C 180,E1 3385.059,E2 3385.059} C_VEL
LIN {X 0,Y 554.304,Z 476.03,A -85,B 0,C 180,E1 3390.939,E2 3390.939} C_VEL
LIN {X 0,Y 554.211,Z 476.03,A -85,B 0,C 180,E1 3397.512,E2 3397.512} C_VEL
LIN {X 0,Y 554.3,Z 476.03,A -85,B 0,C 180,E1 3401.239,E2 3401.239} C_VEL
LIN {X 0,Y 557.539,Z 499.113,A -85,B 0,C 180,E1 3401.861,E2 3401.861} C_VEL
LIN {X 0,Y 556.963,Z 528.543,A -85,B 0,C 180,E1 3403.007,E2 3403.007} C_VEL
LIN {X 0,Y 556.309,Z 557.755,A -85,B 0,C 180,E1 3404.843,E2 3404.843} C_VEL
LIN {X 0,Y 555.636,Z 583.089,A -85,B 0,C 180,E1 3407.207,E2 3407.207} C_VEL
LIN {X 0,Y 555.199,Z 603.59,A -85,B 0,C 180,E1 3409.986,E2 3409.986} C_VEL
LIN {X 0,Y 554.95,Z 618.215,A -85,B 0,C 180,E1 3412.946,E2 3412.946} C_VEL
LIN {X 0,Y 554.882,Z 627.527,A -85,B 0,C 180,E1 3416.086,E2 3416.086} C_VEL
LIN {X 0,Y 554.804,Z 630.887,A -85,B 0,C 180,E1 3418.434,E2 3418.434} C_VEL
LIN {X 0,Y 554.804,Z 630.807,A -85,B 0,C 180,E1 3421.561,E2 3421.561} C_VEL
LIN {X 0,Y 554.866,Z 625.537,A -85,B 0,C 180,E1 3424.693,E2 3424.693} C_VEL
LIN {X 0,Y 554.972,Z 614.54,A -85,B 0,C 180,E1 3427.837,E2 3427.837} C_VEL
LIN {X 0,Y 555.319,Z 597.592,A -85,B 0,C 180,E1 3430.849,E2 3430.849} C_VEL
LIN {X 0,Y 555.782,Z 576.687,A -85,B 0,C 180,E1 3433.386,E2 3433.386} C_VEL
LIN {X 0,Y 556.317,Z 556.958,A -85,B 0,C 180,E1 3435.126,E2 3435.126} C_VEL
LIN {X 0,Y 552.869,Z 543.222,A -85,B 0,C 180,E1 3436.199,E2 3436.199} C_VEL
LIN {X 0,Y 549.486,Z 530.637,A -85,B 0,C 180,E1 3437.038,E2 3437.038} C_VEL
LIN {X 0,Y 549.451,Z 528.654,A -85,B 0,C 180,E1 3437.141,E2 3437.141} C_VEL
LIN {X 0,Y 550.052,Z 497.699,A -85,B 0,C 180,E1 3438.325,E2 3438.325} C_VEL
LIN {X 0,Y 548.799,Z 485.141,A -85,B 0,C 180,E1 3438.655,E2 3438.655} C_VEL
LIN {X 0,Y 546.579,Z 476.03,A -85,B 0,C 180,E1 3438.961,E2 3438.961} C_VEL
LIN {X 0,Y 546.357,Z 476.03,A -85,B 0,C 180,E1 3444.558,E2 3444.558} C_VEL
LIN {X 0,Y 546.119,Z 476.03,A -85,B 0,C 180,E1 3450.742,E2 3450.742} C_VEL
LIN {X 0,Y 546.142,Z 476.03,A -85,B 0,C 180,E1 3456.487,E2 3456.487} C_VEL
LIN {X 0,Y 546.226,Z 476.03,A -85,B 0,C 180,E1 3461.696,E2 3461.696} C_VEL
LIN {X 0,Y 546.169,Z 476.03,A -85,B 0,C 180,E1 3466.127,E2 3466.127} C_VEL
LIN {X 0,Y 546.124,Z 476.03,A -85,B 0,C 180,E1 3472.414,E2 3472.414} C_VEL
LIN {X 0,Y 546.405,Z 476.629,A -85,B 0,C 180,E1 3476.729,E2 3476.729} C_VEL
LIN {X 0,Y 555.941,Z 498.25,A -85,B 0,C 180,E1 3477.696,E2 3477.696} C_VEL
LIN {X 0,Y 555.662,Z 550.195,A -85,B 0,C 180,E1 3478.633,E2 3478.633} C_VEL
LIN {X 0,Y 554.508,Z 589.109,A -85,B 0,C 180,E1 3479.959,E2 3479.959} C_VEL
LIN {X 0,Y 552.86,Z 626.449,A -85,B 0,C 180,E1 3481.882,E2 3481.882} C_VEL
LIN {X 0,Y 551.146,Z 662.098,A -85,B 0,C 180,E1 3484.444,E2 3484.444} C_VEL
LIN {X 0,Y 549.514,Z 694.213,A -85,B 0,C 180,E1 3487.527,E2 3487.527} C_VEL
LIN {X 0,Y 548.36,Z 722.172,A -85,B 0,C 180,E1 3491.068,E2 3491.068} C_VEL
LIN {X 0,Y 547.562,Z 745.268,A -85,B 0,C 180,E1 3494.966,E2 3494.966} C_VEL
LIN {X 0,Y 547.07,Z 762.98,A -85,B 0,C 180,E1 3499.14,E2 3499.14} C_VEL
LIN {X 0,Y 546.929,Z 773.55,A -85,B 0,C 180,E1 3502.843,E2 3502.843} C_VEL
LIN {X 0,Y 546.793,Z 779.917,A -85,B 0,C 180,E1 3506.825,E2 3506.825} C_VEL
LIN {X 0,Y 546.794,Z 781.5,A -85,B 0,C 180,E1 3510,E2 3510} C_VEL
LIN {X 0,Y 546.862,Z 779.918,A -85,B 0,C 180,E1 3513.174,E2 3513.174} C_VEL
LIN {X 0,Y 546.971,Z 773.551,A -85,B 0,C 180,E1 3517.156,E2 3517.156} C_VEL
LIN {X 0,Y 547.143,Z 761.901,A -85,B 0,C 180,E1 3521.169,E2 3521.169} C_VEL
LIN {X 0,Y 547.596,Z 743.515,A -85,B 0,C 180,E1 3525.372,E2 3525.372} C_VEL
LIN {X 0,Y 548.408,Z 720.731,A -85,B 0,C 180,E1 3529.139,E2 3529.139} C_VEL
LIN {X 0,Y 549.579,Z 694.184,A -85,B 0,C 180,E1 3532.474,E2 3532.474} C_VEL
LIN {X 0,Y 551.191,Z 662.148,A -85,B 0,C 180,E1 3535.55,E2 3535.55} C_VEL
LIN {X 0,Y 552.896,Z 626.25,A -85,B 0,C 180,E1 3538.129,E2 3538.129} C_VEL
LIN {X 0,Y 554.525,Z 587.538,A -85,B 0,C 180,E1 3540.109,E2 3540.109} C_VEL
LIN {X 0,Y 555.816,Z 548.527,A -85,B 0,C 180,E1 3541.401,E2 3541.401} C_VEL
LIN {X 0,Y 555.286,Z 496.52,A -85,B 0,C 180,E1 3542.373,E2 3542.373} C_VEL
LIN {X 0,Y 546.151,Z 476.03,A -85,B 0,C 180,E1 3543.33,E2 3543.33} C_VEL
LIN {X 0,Y 546.185,Z 476.03,A -85,B 0,C 180,E1 3549.613,E2 3549.613} C_VEL
LIN {X 0,Y 546.193,Z 476.03,A -85,B 0,C 180,E1 3553.891,E2 3553.891} C_VEL
LIN {X 0,Y 546.102,Z 476.03,A -85,B 0,C 180,E1 3560.386,E2 3560.386} C_VEL
LIN {X 0,Y 546.239,Z 476.03,A -85,B 0,C 180,E1 3566.338,E2 3566.338} C_VEL
LIN {X 0,Y 546.216,Z 476.03,A -85,B 0,C 180,E1 3571.89,E2 3571.89} C_VEL
LIN {X 0,Y 546.242,Z 476.03,A -85,B 0,C 180,E1 3577.17,E2 3577.17} C_VEL
LIN {X 0,Y 546.423,Z 476.03,A -85,B 0,C 180,E1 3582.257,E2 3582.257} C_VEL
LIN {X 0,Y 546.492,Z 476.03,A -85,B 0,C 180,E1 3587.198,E2 3587.198} C_VEL
LIN {X 0,Y 546.534,Z 476.03,A -85,B 0,C 180,E1 3592.041,E2 3592.041} C_VEL
LIN {X 0,Y 546.711,Z 476.03,A -85,B 0,C 180,E1 3596.827,E2 3596.827} C_VEL
LIN {X 0,Y 546.788,Z 476.03,A -85,B 0,C 180,E1 3601.589,E2 3601.589} C_VEL
LIN {X 0,Y 546.722,Z 476.03,A -85,B 0,C 180,E1 3606.362,E2 3606.362} C_VEL
LIN {X 0,Y 546.39,Z 476.03,A -85,B 0,C 180,E1 3612.81,E2 3612.81} C_VEL
LIN {X 0,Y 546.351,Z 476.03,A -85,B 0,C 180,E1 3617.75,E2 3617.75} C_VEL
LIN {X 0,Y 546.333,Z 476.03,A -85,B 0,C 180,E1 3622.831,E2 3622.831} C_VEL
LIN {X 0,Y 546.254,Z 476.03,A -85,B 0,C 180,E1 3628.113,E2 3628.113} C_VEL
LIN {X 0,Y 546.147,Z 476.03,A -85,B 0,C 180,E1 3633.726,E2 3633.726} C_VEL
LIN {X 0,Y 546.227,Z 476.03,A -85,B 0,C 180,E1 3639.609,E2 3639.609} C_VEL
LIN {X 0,Y 546.227,Z 476.03,A -85,B 0,C 180,E1 3646.133,E2 3646.133} C_VEL
LIN {X 0,Y 546.188,Z 476.03,A -85,B 0,C 180,E1 3652.42,E2 3652.42} C_VEL
LIN {X 0,Y 546.145,Z 476.03,A -85,B 0,C 180,E1 3658.214,E2 3658.214} C_VEL
LIN {X 0,Y 546.308,Z 476.03,A -85,B 0,C 180,E1 3663.676,E2 3663.676} C_VEL
LIN {X 0,Y 546.416,Z 476.03,A -85,B 0,C 180,E1 3668.886,E2 3668.886} C_VEL
LIN {X 0,Y 546.371,Z 476.052,A -85,B 0,C 180,E1 3674.88,E2 3674.88} C_VEL
LIN {X 0,Y 555.013,Z 500.977,A -85,B 0,C 180,E1 3676.209,E2 3676.209} C_VEL
LIN {X 0,Y 553.549,Z 541.08,A -85,B 0,C 180,E1 3677.962,E2 3677.962} C_VEL
LIN {X 0,Y 551.913,Z 577.086,A -85,B 0,C 180,E1 3680.227,E2 3680.227} C_VEL
LIN {X 0,Y 550.247,Z 610.769,A -85,B 0,C 180,E1 3683.086,E2 3683.086} C_VEL
LIN {X 0,Y 548.809,Z 640.605,A -85,B 0,C 180,E1 3686.441,E2 3686.441} C_VEL
LIN {X 0,Y 547.811,Z 664.723,A -85,B 0,C 180,E1 3690,E2 3690} C_VEL
LIN {X 0,Y 547.295,Z 683.024,A -85,B 0,C 180,E1 3693.569,E2 3693.569} C_VEL
LIN {X 0,Y 547.01,Z 697.664,A -85,B 0,C 180,E1 3697.555,E2 3697.555} C_VEL
LIN {X 0,Y 546.888,Z 706.303,A -85,B 0,C 180,E1 3701.175,E2 3701.175} C_VEL
LIN {X 0,Y 546.722,Z 710.482,A -85,B 0,C 180,E1 3704.433,E2 3704.433} C_VEL
LIN {X 0,Y 546.673,Z 711.342,A -85,B 0,C 180,E1 3707.738,E2 3707.738} C_VEL
LIN {X 0,Y 546.762,Z 708.82,A -85,B 0,C 180,E1 3711.101,E2 3711.101} C_VEL
LIN {X 0,Y 546.922,Z 700.645,A -85,B 0,C 180,E1 3715.311,E2 3715.311} C_VEL
LIN {X 0,Y 547.207,Z 686.259,A -85,B 0,C 180,E1 3719.589,E2 3719.589} C_VEL
LIN {X 0,Y 547.755,Z 666.741,A -85,B 0,C 180,E1 3723.563,E2 3723.563} C_VEL
LIN {X 0,Y 548.712,Z 642.576,A -85,B 0,C 180,E1 3727.215,E2 3727.215} C_VEL
LIN {X 0,Y 550.136,Z 612.293,A -85,B 0,C 180,E1 3730.672,E2 3730.672} C_VEL
LIN {X 0,Y 551.795,Z 579.427,A -85,B 0,C 180,E1 3733.508,E2 3733.508} C_VEL
LIN {X 0,Y 553.532,Z 542.772,A -85,B 0,C 180,E1 3735.858,E2 3735.858} C_VEL
LIN {X 0,Y 555.037,Z 504.158,A -85,B 0,C 180,E1 3737.583,E2 3737.583} C_VEL
LIN {X 0,Y 554.079,Z 496.936,A -85,B 0,C 180,E1 3737.897,E2 3737.897} C_VEL
LIN {X 0,Y 546.114,Z 476.03,A -85,B 0,C 180,E1 3739.114,E2 3739.114} C_VEL
LIN {X 0,Y 546.118,Z 476.03,A -85,B 0,C 180,E1 3744.393,E2 3744.393} C_VEL
LIN {X 0,Y 546.301,Z 476.03,A -85,B 0,C 180,E1 3750.073,E2 3750.073} C_VEL
LIN {X 0,Y 546.237,Z 476.03,A -85,B 0,C 180,E1 3756.168,E2 3756.168} C_VEL
LIN {X 0,Y 546.371,Z 476.03,A -85,B 0,C 180,E1 3760.989,E2 3760.989} C_VEL
LIN {X 0,Y 550.056,Z 498.149,A -85,B 0,C 180,E1 3761.588,E2 3761.588} C_VEL
LIN {X 0,Y 549.366,Z 528.63,A -85,B 0,C 180,E1 3762.764,E2 3762.764} C_VEL
LIN {X 0,Y 548.629,Z 556.38,A -85,B 0,C 180,E1 3764.516,E2 3764.516} C_VEL
LIN {X 0,Y 547.91,Z 581.265,A -85,B 0,C 180,E1 3766.82,E2 3766.82} C_VEL
LIN {X 0,Y 547.409,Z 601.465,A -85,B 0,C 180,E1 3769.498,E2 3769.498} C_VEL
LIN {X 0,Y 547.102,Z 616.632,A -85,B 0,C 180,E1 3772.444,E2 3772.444} C_VEL
LIN {X 0,Y 547.026,Z 625.741,A -85,B 0,C 180,E1 3775.235,E2 3775.235} C_VEL
LIN {X 0,Y 546.902,Z 630.885,A -85,B 0,C 180,E1 3778.411,E2 3778.411} C_VEL
LIN {X 0,Y 546.903,Z 630.806,A -85,B 0,C 180,E1 3781.584,E2 3781.584} C_VEL
LIN {X 0,Y 546.972,Z 625.541,A -85,B 0,C 180,E1 3784.761,E2 3784.761} C_VEL
LIN {X 0,Y 547.122,Z 614.544,A -85,B 0,C 180,E1 3787.951,E2 3787.951} C_VEL
LIN {X 0,Y 547.489,Z 597.598,A -85,B 0,C 180,E1 3791.006,E2 3791.006} C_VEL
LIN {X 0,Y 548.028,Z 576.691,A -85,B 0,C 180,E1 3793.579,E2 3793.579} C_VEL
LIN {X 0,Y 548.876,Z 550.208,A -85,B 0,C 180,E1 3795.852,E2 3795.852} C_VEL
LIN {X 0,Y 549.451,Z 528.654,A -85,B 0,C 180,E1 3797.141,E2 3797.141} C_VEL
LIN {X 0,Y 546.045,Z 513.22,A -85,B 0,C 180,E1 3797.94,E2 3797.94} C_VEL
LIN {X 0,Y 542.542,Z 499.308,A -85,B 0,C 180,E1 3798.513,E2 3798.513} C_VEL
LIN {X 0,Y 542.484,Z 497.198,A -85,B 0,C 180,E1 3798.573,E2 3798.573} C_VEL
LIN {X 0,Y 540.618,Z 484.442,A -85,B 0,C 180,E1 3798.91,E2 3798.91} C_VEL
LIN {X 0,Y 538.652,Z 476.03,A -85,B 0,C 180,E1 3799.16,E2 3799.16} C_VEL
LIN {X 0,Y 538.402,Z 476.03,A -85,B 0,C 180,E1 3804.946,E2 3804.946} C_VEL
LIN {X 0,Y 538.232,Z 476.03,A -85,B 0,C 180,E1 3810.417,E2 3810.417} C_VEL
LIN {X 0,Y 538.222,Z 476.03,A -85,B 0,C 180,E1 3816.205,E2 3816.205} C_VEL
LIN {X 0,Y 538.233,Z 476.03,A -85,B 0,C 180,E1 3822.459,E2 3822.459} C_VEL
LIN {X 0,Y 538.156,Z 476.03,A -85,B 0,C 180,E1 3827.526,E2 3827.526} C_VEL
LIN {X 0,Y 538.207,Z 476.03,A -85,B 0,C 180,E1 3833.787,E2 3833.787} C_VEL
LIN {X 0,Y 538.376,Z 476.03,A -85,B 0,C 180,E1 3836.144,E2 3836.144} C_VEL
LIN {X 0,Y 549.257,Z 500.345,A -85,B 0,C 180,E1 3837.286,E2 3837.286} C_VEL
LIN {X 0,Y 548.908,Z 550.183,A -85,B 0,C 180,E1 3838.202,E2 3838.202} C_VEL
LIN {X 0,Y 547.637,Z 588.374,A -85,B 0,C 180,E1 3839.509,E2 3839.509} C_VEL
LIN {X 0,Y 545.869,Z 624.733,A -85,B 0,C 180,E1 3841.379,E2 3841.379} C_VEL
LIN {X 0,Y 543.995,Z 659.503,A -85,B 0,C 180,E1 3843.859,E2 3843.859} C_VEL
LIN {X 0,Y 542.144,Z 692.265,A -85,B 0,C 180,E1 3846.983,E2 3846.983} C_VEL
LIN {X 0,Y 540.744,Z 719.261,A -85,B 0,C 180,E1 3850.366,E2 3850.366} C_VEL
LIN {X 0,Y 539.749,Z 742.092,A -85,B 0,C 180,E1 3854.127,E2 3854.127} C_VEL
LIN {X 0,Y 539.19,Z 758.852,A -85,B 0,C 180,E1 3857.842,E2 3857.842} C_VEL
LIN {X 0,Y 539.052,Z 770.64,A -85,B 0,C 180,E1 3861.52,E2 3861.52} C_VEL
LIN {X 0,Y 538.913,Z 777.955,A -85,B 0,C 180,E1 3865.165,E2 3865.165} C_VEL
LIN {X 0,Y 538.888,Z 781.101,A -85,B 0,C 180,E1 3868.39,E2 3868.39} C_VEL
LIN {X 0,Y 539.028,Z 781.101,A -85,B 0,C 180,E1 3871.609,E2 3871.609} C_VEL
LIN {X 0,Y 538.89,Z 776.716,A -85,B 0,C 180,E1 3875.643,E2 3875.643} C_VEL
LIN {X 0,Y 539.074,Z 767.232,A -85,B 0,C 180,E1 3879.702,E2 3879.702} C_VEL
LIN {X 0,Y 539.439,Z 752.136,A -85,B 0,C 180,E1 3883.795,E2 3883.795} C_VEL
LIN {X 0,Y 540.2,Z 732.077,A -85,B 0,C 180,E1 3887.661,E2 3887.661} C_VEL
LIN {X 0,Y 541.519,Z 705.215,A -85,B 0,C 180,E1 3891.506,E2 3891.506} C_VEL
LIN {X 0,Y 543.116,Z 675.569,A -85,B 0,C 180,E1 3894.719,E2 3894.719} C_VEL
LIN {X 0,Y 544.909,Z 641.896,A -85,B 0,C 180,E1 3897.492,E2 3897.492} C_VEL
LIN {X 0,Y 546.863,Z 604.368,A -85,B 0,C 180,E1 3899.751,E2 3899.751} C_VEL
LIN {X 0,Y 548.377,Z 565.251,A -85,B 0,C 180,E1 3901.36,E2 3901.36} C_VEL
LIN {X 0,Y 549.517,Z 525.701,A -85,B 0,C 180,E1 3902.302,E2 3902.302} C_VEL
LIN {X 0,Y 548.603,Z 499.042,A -85,B 0,C 180,E1 3902.778,E2 3902.778} C_VEL
LIN {X 0,Y 538.224,Z 476.03,A -85,B 0,C 180,E1 3903.904,E2 3903.904} C_VEL
LIN {X 0,Y 538.28,Z 476.03,A -85,B 0,C 180,E1 3908.231,E2 3908.231} C_VEL
LIN {X 0,Y 538.207,Z 476.03,A -85,B 0,C 180,E1 3914.693,E2 3914.693} C_VEL
LIN {X 0,Y 538.136,Z 476.03,A -85,B 0,C 180,E1 3919.681,E2 3919.681} C_VEL
LIN {X 0,Y 538.262,Z 476.03,A -85,B 0,C 180,E1 3925.77,E2 3925.77} C_VEL
LIN {X 0,Y 538.272,Z 476.03,A -85,B 0,C 180,E1 3931.437,E2 3931.437} C_VEL
LIN {X 0,Y 538.332,Z 476.03,A -85,B 0,C 180,E1 3936.816,E2 3936.816} C_VEL
LIN {X 0,Y 538.491,Z 476.03,A -85,B 0,C 180,E1 3942.94,E2 3942.94} C_VEL
LIN {X 0,Y 538.525,Z 476.03,A -85,B 0,C 180,E1 3948.653,E2 3948.653} C_VEL
LIN {X 0,Y 538.593,Z 476.03,A -85,B 0,C 180,E1 3953.546,E2 3953.546} C_VEL
LIN {X 0,Y 538.669,Z 476.03,A -85,B 0,C 180,E1 3958.392,E2 3958.392} C_VEL
LIN {X 0,Y 538.644,Z 476.03,A -85,B 0,C 180,E1 3963.225,E2 3963.225} C_VEL
LIN {X 0,Y 538.534,Z 476.03,A -85,B 0,C 180,E1 3968.083,E2 3968.083} C_VEL
LIN {X 0,Y 538.497,Z 476.03,A -85,B 0,C 180,E1 3973.001,E2 3973.001} C_VEL
LIN {X 0,Y 538.448,Z 476.03,A -85,B 0,C 180,E1 3978.019,E2 3978.019} C_VEL
LIN {X 0,Y 538.426,Z 476.03,A -85,B 0,C 180,E1 3983.186,E2 3983.186} C_VEL
LIN {X 0,Y 538.287,Z 476.03,A -85,B 0,C 180,E1 3988.567,E2 3988.567} C_VEL
LIN {X 0,Y 538.22,Z 476.03,A -85,B 0,C 180,E1 3994.239,E2 3994.239} C_VEL
LIN {X 0,Y 538.348,Z 476.03,A -85,B 0,C 180,E1 3998.225,E2 3998.225} C_VEL
LIN {X 0,Y 538.228,Z 476.03,A -85,B 0,C 180,E1 4004.691,E2 4004.691} C_VEL
LIN {X 0,Y 538.235,Z 476.03,A -85,B 0,C 180,E1 4009.683,E2 4009.683} C_VEL
LIN {X 0,Y 538.155,Z 476.03,A -85,B 0,C 180,E1 4015.757,E2 4015.757} C_VEL
LIN {X 0,Y 538.261,Z 476.03,A -85,B 0,C 180,E1 4021.432,E2 4021.432} C_VEL
LIN {X 0,Y 538.409,Z 476.03,A -85,B 0,C 180,E1 4026.815,E2 4026.815} C_VEL
LIN {X 0,Y 538.512,Z 476.03,A -85,B 0,C 180,E1 4031.984,E2 4031.984} C_VEL
LIN {X 0,Y 538.481,Z 476.19,A -85,B 0,C 180,E1 4034.356,E2 4034.356} C_VEL
LIN {X 0,Y 548.133,Z 502.457,A -85,B 0,C 180,E1 4035.834,E2 4035.834} C_VEL
LIN {X 0,Y 546.435,Z 543.859,A -85,B 0,C 180,E1 4037.701,E2 4037.701} C_VEL
LIN {X 0,Y 544.532,Z 580.362,A -85,B 0,C 180,E1 4040.093,E2 4040.093} C_VEL
LIN {X 0,Y 542.747,Z 612.04,A -85,B 0,C 180,E1 4042.868,E2 4042.868} C_VEL
LIN {X 0,Y 541.122,Z 642.518,A -85,B 0,C 180,E1 4046.391,E2 4046.391} C_VEL
LIN {X 0,Y 539.977,Z 667.302,A -85,B 0,C 180,E1 4050.201,E2 4050.201} C_VEL
LIN {X 0,Y 539.36,Z 685.485,A -85,B 0,C 180,E1 4053.949,E2 4053.949} C_VEL
LIN {X 0,Y 539.05,Z 699.516,A -85,B 0,C 180,E1 4058.074,E2 4058.074} C_VEL
LIN {X 0,Y 538.889,Z 708.026,A -85,B 0,C 180,E1 4062.165,E2 4062.165} C_VEL
LIN {X 0,Y 538.77,Z 711.374,A -85,B 0,C 180,E1 4066.322,E2 4066.322} C_VEL
LIN {X 0,Y 538.814,Z 710.333,A -85,B 0,C 180,E1 4069.707,E2 4069.707} C_VEL
LIN {X 0,Y 538.985,Z 704.592,A -85,B 0,C 180,E1 4073.723,E2 4073.723} C_VEL
LIN {X 0,Y 539.234,Z 692.744,A -85,B 0,C 180,E1 4078.037,E2 4078.037} C_VEL
LIN {X 0,Y 539.775,Z 675.248,A -85,B 0,C 180,E1 4082.206,E2 4082.206} C_VEL
LIN {X 0,Y 540.671,Z 652.01,A -85,B 0,C 180,E1 4086.189,E2 4086.189} C_VEL
LIN {X 0,Y 542.073,Z 624.114,A -85,B 0,C 180,E1 4089.766,E2 4089.766} C_VEL
LIN {X 0,Y 543.811,Z 593.281,A -85,B 0,C 180,E1 4092.773,E2 4092.773} C_VEL
LIN {X 0,Y 545.699,Z 558.435,A -85,B 0,C 180,E1 4095.346,E2 4095.346} C_VEL
LIN {X 0,Y 547.479,Z 520.555,A -85,B 0,C 180,E1 4097.35,E2 4097.35} C_VEL
LIN {X 0,Y 547.663,Z 500.737,A -85,B 0,C 180,E1 4098.166,E2 4098.166} C_VEL
LIN {X 0,Y 538.177,Z 476.03,A -85,B 0,C 180,E1 4099.678,E2 4099.678} C_VEL
LIN {X 0,Y 538.267,Z 476.03,A -85,B 0,C 180,E1 4105.765,E2 4105.765} C_VEL
LIN {X 0,Y 538.327,Z 476.03,A -85,B 0,C 180,E1 4111.435,E2 4111.435} C_VEL
LIN {X 0,Y 538.342,Z 476.03,A -85,B 0,C 180,E1 4116.811,E2 4116.811} C_VEL
LIN {X 0,Y 538.42,Z 476.03,A -85,B 0,C 180,E1 4120.747,E2 4120.747} C_VEL
LIN {X 0,Y 542.519,Z 497.582,A -85,B 0,C 180,E1 4121.326,E2 4121.326} C_VEL
LIN {X 0,Y 541.8,Z 528.779,A -85,B 0,C 180,E1 4122.516,E2 4122.516} C_VEL
LIN {X 0,Y 541.015,Z 557.175,A -85,B 0,C 180,E1 4124.311,E2 4124.311} C_VEL
LIN {X 0,Y 540.197,Z 581.742,A -85,B 0,C 180,E1 4126.628,E2 4126.628} C_VEL
LIN {X 0,Y 539.594,Z 601.385,A -85,B 0,C 180,E1 4129.323,E2 4129.323} C_VEL
LIN {X 0,Y 539.228,Z 616.627,A -85,B 0,C 180,E1 4132.333,E2 4132.333} C_VEL
LIN {X 0,Y 539.103,Z 626.505,A -85,B 0,C 180,E1 4135.491,E2 4135.491} C_VEL
LIN {X 0,Y 539.016,Z 630.882,A -85,B 0,C 180,E1 4138.388,E2 4138.388} C_VEL
LIN {X 0,Y 539.016,Z 630.804,A -85,B 0,C 180,E1 4141.607,E2 4141.607} C_VEL
LIN {X 0,Y 539.08,Z 625.545,A -85,B 0,C 180,E1 4144.831,E2 4144.831} C_VEL
